LIN {X 0.027,Y -509.372,Z 664.122,A 0.000,B 0.000,C 90.000,E1 237.995} C_DIS
LIN {X 0.006,Y -505.336,Z 664.112,A 0.000,B 0.000,C 90.000,E1 236.215} C_DIS
LIN {X -0.007,Y -502.437,Z 664.106,A 0.000,B 0.000,C 90.000,E1 235.022} C_DIS
LIN {X 0.219,Y -498.643,Z 664.097,A 0.000,B 0.000,C 90.000,E1 233.497} C_DIS
LIN {X -0.007,Y -491.952,Z 664.082,A 0.000,B 0.000,C 90.000,E1 230.803} C_DIS
LIN {X -0.006,Y -487.620,Z 664.072,A 0.000,B 0.000,C 90.000,E1 228.976} C_DIS
LIN {X 0.039,Y -482.507,Z 664.060,A 0.000,B 0.000,C 90.000,E1 226.824} C_DIS
LIN {X 0.020,Y -478.874,Z 664.052,A 0.000,B 0.000,C 90.000,E1 225.283} C_DIS
LIN {X 0.140,Y -473.719,Z 664.040,A 0.000,B 0.000,C 90.000,E1 223.095} C_DIS
LIN {X -0.036,Y -467.402,Z 664.024,A 0.000,B 0.000,C 90.000,E1 220.297} C_DIS
LIN {X 0.130,Y -463.516,Z 664.013,A 0.000,B 0.000,C 90.000,E1 218.382} C_DIS
LIN {X 0.034,Y -459.004,Z 664.001,A 0.000,B 0.000,C 90.000,E1 216.171} C_DIS
LIN {X 0.087,Y -455.266,Z 663.990,A 0.000,B 0.000,C 90.000,E1 214.246} C_DIS
LIN {X 0.106,Y -452.881,Z 663.983,A 0.000,B 0.000,C 90.000,E1 212.959} C_DIS
LIN {X -0.122,Y -449.264,Z 663.972,A 0.000,B 0.000,C 90.000,E1 211.052} C_DIS
LIN {X 0.103,Y -445.713,Z 663.962,A 0.000,B 0.000,C 90.000,E1 209.077} C_DIS
LIN {X -0.017,Y -442.739,Z 663.953,A 0.000,B 0.000,C 90.000,E1 207.462} C_DIS
LIN {X -0.194,Y -439.843,Z 663.943,A 0.000,B 0.000,C 90.000,E1 205.848} C_DIS
LIN {X -0.225,Y -436.925,Z 663.934,A 0.000,B 0.000,C 90.000,E1 204.207} C_DIS
LIN {X -0.094,Y -433.311,Z 663.923,A 0.000,B 0.000,C 90.000,E1 202.206} C_DIS
LIN {X -0.011,Y -429.068,Z 663.910,A 0.000,B 0.000,C 90.000,E1 199.866} C_DIS
LIN {X -0.132,Y -425.619,Z 663.899,A 0.000,B 0.000,C 90.000,E1 197.873} C_DIS
LIN {X -0.234,Y -422.836,Z 663.890,A 0.000,B 0.000,C 90.000,E1 196.205} C_DIS
LIN {X 0.185,Y -419.483,Z 663.879,A 0.000,B 0.000,C 90.000,E1 194.120} C_DIS
LIN {X -0.098,Y -416.086,Z 663.867,A 0.000,B 0.000,C 90.000,E1 192.119} C_DIS
LIN {X -0.141,Y -412.932,Z 663.856,A 0.000,B 0.000,C 90.000,E1 190.074} C_DIS
LIN {X 0.011,Y -409.838,Z 663.844,A 0.000,B 0.000,C 90.000,E1 187.992} C_DIS
LIN {X 0.058,Y -406.301,Z 663.831,A 0.000,B 0.000,C 90.000,E1 185.568} C_DIS
LIN {X -0.081,Y -402.738,Z 663.816,A 0.000,B 0.000,C 90.000,E1 182.808} C_DIS
LIN {X -0.038,Y -399.329,Z 663.798,A 0.000,B 0.000,C 90.000,E1 179.656} C_DIS
LIN {X -0.157,Y -396.563,Z 663.779,A 0.000,B 0.000,C 90.000,E1 176.159} C_DIS
LIN {X 0.204,Y -394.877,Z 663.761,A 0.000,B 0.000,C 90.000,E1 172.932} C_DIS
LIN {X -0.093,Y -394.008,Z 663.747,A 0.000,B 0.000,C 90.000,E1 170.500} C_DIS
LIN {X 0.062,Y -393.548,Z 663.731,A 0.000,B 0.000,C 90.000,E1 167.645} C_DIS
LIN {X 0.067,Y -393.374,Z 663.720,A 0.000,B 0.000,C 90.000,E1 165.519} C_DIS
LIN {X 0.114,Y -393.447,Z 663.706,A 0.000,B 0.000,C 90.000,E1 163.032} C_DIS
LIN {X 0.127,Y -393.772,Z 663.692,A 0.000,B 0.000,C 90.000,E1 160.550} C_DIS
LIN {X -0.021,Y -393.961,Z 663.684,A 0.000,B 0.000,C 90.000,E1 159.156} C_DIS
LIN {X -0.140,Y -394.297,Z 663.672,A 0.000,B 0.000,C 90.000,E1 157.050} C_DIS
LIN {X -0.030,Y -394.820,Z 663.657,A 0.000,B 0.000,C 90.000,E1 154.204} C_DIS
LIN {X 0.159,Y -395.196,Z 663.647,A 0.000,B 0.000,C 90.000,E1 152.410} C_DIS
LIN {X -0.136,Y -395.685,Z 663.635,A 0.000,B 0.000,C 90.000,E1 150.333} C_DIS
LIN {X -0.161,Y -396.344,Z 663.621,A 0.000,B 0.000,C 90.000,E1 147.867} C_DIS
LIN {X -0.079,Y -397.264,Z 663.608,A 0.000,B 0.000,C 90.000,E1 145.388} C_DIS
LIN {X 0.066,Y -398.259,Z 663.596,A 0.000,B 0.000,C 90.000,E1 143.256} C_DIS
LIN {X -0.084,Y -399.368,Z 663.584,A 0.000,B 0.000,C 90.000,E1 141.170} C_DIS
LIN {X 0.099,Y -400.918,Z 663.571,A 0.000,B 0.000,C 90.000,E1 138.690} C_DIS
LIN {X -0.036,Y -401.754,Z 663.563,A 0.000,B 0.000,C 90.000,E1 137.310} C_DIS
LIN {X 0.162,Y -403.361,Z 663.549,A 0.000,B 0.000,C 90.000,E1 134.838} C_DIS
LIN {X -0.124,Y -404.797,Z 663.540,A 0.000,B 0.000,C 90.000,E1 133.137} C_DIS
LIN {X -0.166,Y -405.700,Z 663.536,A 0.000,B 0.000,C 90.000,E1 132.447} C_DIS
LIN {X -0.200,Y -406.988,Z 663.532,A 0.000,B 0.000,C 90.000,E1 131.757} C_DIS
LIN {X -0.183,Y -409.105,Z 663.529,A 0.000,B 0.000,C 90.000,E1 131.148} C_DIS
LIN {X -0.042,Y -411.236,Z 663.527,A 0.000,B 0.000,C 90.000,E1 130.782} C_DIS
LIN {X -0.120,Y -412.190,Z 663.526,A 0.000,B 0.000,C 90.000,E1 130.620} C_DIS
LIN {X -0.196,Y -413.918,Z 663.525,A 0.000,B 0.000,C 90.000,E1 130.458} C_DIS
LIN {X 0.055,Y -417.079,Z 663.523,A 0.000,B 0.000,C 90.000,E1 130.092} C_DIS
LIN {X -0.146,Y -423.546,Z 663.520,A 0.000,B 0.000,C 90.000,E1 129.564} C_DIS
LIN {X 0.122,Y -449.130,Z 663.509,A 0.000,B 0.000,C 90.000,E1 127.604} C_DIS
LIN {X 0.249,Y -459.985,Z 663.505,A 0.000,B 0.000,C 90.000,E1 126.790} C_DIS
LIN {X 0.184,Y -467.766,Z 663.501,A 0.000,B 0.000,C 90.000,E1 126.217} C_DIS
LIN {X 0.030,Y -473.899,Z 663.499,A 0.000,B 0.000,C 90.000,E1 125.758} C_DIS
LIN {X 0.100,Y -481.253,Z 663.495,A 0.000,B 0.000,C 90.000,E1 125.152} C_DIS
LIN {X -0.243,Y -485.709,Z 663.493,A 0.000,B 0.000,C 90.000,E1 124.818} C_DIS
LIN {X 0.011,Y -491.516,Z 663.490,A 0.000,B 0.000,C 90.000,E1 124.278} C_DIS
LIN {X 0.140,Y -500.006,Z 663.486,A 0.000,B 0.000,C 90.000,E1 123.499} C_DIS
LIN {X -0.253,Y -509.537,Z 663.481,A 0.000,B 0.000,C 90.000,E1 122.625} C_DIS
LIN {X -0.014,Y -515.907,Z 663.478,A 0.000,B 0.000,C 90.000,E1 121.957} C_DIS
LIN {X 0.036,Y -523.749,Z 663.473,A 0.000,B 0.000,C 90.000,E1 121.131} C_DIS
LIN {X -0.228,Y -528.777,Z 663.470,A 0.000,B 0.000,C 90.000,E1 120.590} C_DIS
LIN {X -0.159,Y -533.124,Z 663.467,A 0.000,B 0.000,C 90.000,E1 120.050} C_DIS
LIN {X -0.017,Y -537.366,Z 663.464,A 0.000,B 0.000,C 90.000,E1 119.461} C_DIS
LIN {X 0.025,Y -542.151,Z 663.460,A 0.000,B 0.000,C 90.000,E1 118.743} C_DIS
LIN {X 0.114,Y -546.377,Z 663.456,A 0.000,B 0.000,C 90.000,E1 118.025} C_DIS
LIN {X 0.105,Y -549.500,Z 663.453,A 0.000,B 0.000,C 90.000,E1 117.462} C_DIS
LIN {X 0.147,Y -553.631,Z 663.448,A 0.000,B 0.000,C 90.000,E1 116.616} C_DIS
LIN {X 0.091,Y -556.868,Z 663.444,A 0.000,B 0.000,C 90.000,E1 115.924} C_DIS
LIN {X 0.197,Y -560.328,Z 663.440,A 0.000,B 0.000,C 90.000,E1 115.079} C_DIS
LIN {X -0.103,Y -564.545,Z 663.433,A 0.000,B 0.000,C 90.000,E1 114.003} C_DIS
LIN {X -0.054,Y -568.273,Z 663.427,A 0.000,B 0.000,C 90.000,E1 112.898} C_DIS
LIN {X -0.078,Y -570.823,Z 663.423,A 0.000,B 0.000,C 90.000,E1 112.078} C_DIS
LIN {X -0.116,Y -572.382,Z 663.420,A 0.000,B 0.000,C 90.000,E1 111.535} C_DIS
LIN {X 0.054,Y -575.058,Z 663.414,A 0.000,B 0.000,C 90.000,E1 110.429} C_DIS
LIN {X 0.258,Y -577.513,Z 663.408,A 0.000,B 0.000,C 90.000,E1 109.322} C_DIS
LIN {X 0.302,Y -579.804,Z 663.402,A 0.000,B 0.000,C 90.000,E1 108.236} C_DIS
LIN {X -0.080,Y -583.716,Z 663.391,A 0.000,B 0.000,C 90.000,E1 106.386} C_DIS
LIN {X 0.281,Y -586.439,Z 663.384,A 0.000,B 0.000,C 90.000,E1 105.009} C_DIS
LIN {X -0.041,Y -589.129,Z 663.376,A 0.000,B 0.000,C 90.000,E1 103.703} C_DIS
LIN {X -0.151,Y -591.244,Z 663.370,A 0.000,B 0.000,C 90.000,E1 102.647} C_DIS
LIN {X 0.183,Y -595.368,Z 663.358,A 0.000,B 0.000,C 90.000,E1 100.489} C_DIS
LIN {X 0.046,Y -598.366,Z 663.350,A 0.000,B 0.000,C 90.000,E1 98.916} C_DIS
LIN {X -0.053,Y -600.257,Z 663.344,A 0.000,B 0.000,C 90.000,E1 97.871} C_DIS
LIN {X 0.022,Y -602.401,Z 663.336,A 0.000,B 0.000,C 90.000,E1 96.549} C_DIS
LIN {X 0.262,Y -603.616,Z 663.332,A 0.000,B 0.000,C 90.000,E1 95.739} C_DIS
LIN {X -0.197,Y -605.551,Z 663.325,A 0.000,B 0.000,C 90.000,E1 94.473} C_DIS
LIN {X -0.062,Y -607.203,Z 663.318,A 0.000,B 0.000,C 90.000,E1 93.154} C_DIS
LIN {X 0.108,Y -608.659,Z 663.310,A 0.000,B 0.000,C 90.000,E1 91.835} C_DIS
LIN {X 0.296,Y -609.771,Z 663.303,A 0.000,B 0.000,C 90.000,E1 90.516} C_DIS
LIN {X 0.205,Y -610.431,Z 663.297,A 0.000,B 0.000,C 90.000,E1 89.484} C_DIS
LIN {X 0.118,Y -610.892,Z 663.292,A 0.000,B 0.000,C 90.000,E1 88.453} C_DIS
LIN {X 0.054,Y -611.171,Z 663.286,A 0.000,B 0.000,C 90.000,E1 87.421} C_DIS
LIN {X -0.001,Y -611.342,Z 663.280,A 0.000,B 0.000,C 90.000,E1 86.388} C_DIS
LIN {X -0.058,Y -611.310,Z 663.274,A 0.000,B 0.000,C 90.000,E1 85.355} C_DIS
LIN {X 0.205,Y -610.994,Z 663.267,A 0.000,B 0.000,C 90.000,E1 84.033} C_DIS
LIN {X 0.191,Y -610.576,Z 663.261,A 0.000,B 0.000,C 90.000,E1 82.996} C_DIS
LIN {X 0.253,Y -610.067,Z 663.255,A 0.000,B 0.000,C 90.000,E1 81.951} C_DIS
LIN {X 0.219,Y -609.190,Z 663.250,A 0.000,B 0.000,C 90.000,E1 80.914} C_DIS
LIN {X 0.031,Y -608.443,Z 663.245,A 0.000,B 0.000,C 90.000,E1 80.151} C_DIS
LIN {X -0.193,Y -606.957,Z 663.238,A 0.000,B 0.000,C 90.000,E1 78.870} C_DIS
LIN {X 0.271,Y -605.274,Z 663.231,A 0.000,B 0.000,C 90.000,E1 77.521} C_DIS
LIN {X -0.204,Y -603.788,Z 663.225,A 0.000,B 0.000,C 90.000,E1 76.520} C_DIS
LIN {X 0.193,Y -601.761,Z 663.218,A 0.000,B 0.000,C 90.000,E1 75.172} C_DIS
LIN {X 0.099,Y -600.497,Z 663.213,A 0.000,B 0.000,C 90.000,E1 74.393} C_DIS
LIN {X 0.288,Y -598.679,Z 663.208,A 0.000,B 0.000,C 90.000,E1 73.323} C_DIS
LIN {X -0.127,Y -596.729,Z 663.202,A 0.000,B 0.000,C 90.000,E1 72.308} C_DIS
LIN {X 0.179,Y -594.711,Z 663.196,A 0.000,B 0.000,C 90.000,E1 71.221} C_DIS
LIN {X -0.216,Y -591.898,Z 663.188,A 0.000,B 0.000,C 90.000,E1 69.934} C_DIS
LIN {X 0.015,Y -589.281,Z 663.183,A 0.000,B 0.000,C 90.000,E1 68.847} C_DIS
LIN {X -0.011,Y -587.181,Z 663.178,A 0.000,B 0.000,C 90.000,E1 68.050} C_DIS
LIN {X 0.165,Y -584.852,Z 663.174,A 0.000,B 0.000,C 90.000,E1 67.230} C_DIS
LIN {X -0.042,Y -581.402,Z 663.168,A 0.000,B 0.000,C 90.000,E1 66.177} C_DIS
LIN {X 0.079,Y -578.533,Z 663.163,A 0.000,B 0.000,C 90.000,E1 65.357} C_DIS
LIN {X 0.169,Y -575.542,Z 663.159,A 0.000,B 0.000,C 90.000,E1 64.537} C_DIS
LIN {X 0.064,Y -571.154,Z 663.153,A 0.000,B 0.000,C 90.000,E1 63.461} C_DIS
LIN {X -0.008,Y -568.900,Z 663.150,A 0.000,B 0.000,C 90.000,E1 62.922} C_DIS
LIN {X -0.025,Y -565.254,Z 663.145,A 0.000,B 0.000,C 90.000,E1 62.103} C_DIS
LIN {X 0.268,Y -561.861,Z 663.141,A 0.000,B 0.000,C 90.000,E1 61.385} C_DIS
LIN {X 0.223,Y -558.151,Z 663.138,A 0.000,B 0.000,C 90.000,E1 60.717} C_DIS
LIN {X -0.031,Y -553.887,Z 663.134,A 0.000,B 0.000,C 90.000,E1 60.049} C_DIS
LIN {X -0.007,Y -550.136,Z 663.131,A 0.000,B 0.000,C 90.000,E1 59.488} C_DIS
LIN {X -0.207,Y -546.031,Z 663.127,A 0.000,B 0.000,C 90.000,E1 58.948} C_DIS
LIN {X -0.029,Y -540.656,Z 663.124,A 0.000,B 0.000,C 90.000,E1 58.280} C_DIS
LIN {X -0.246,Y -535.968,Z 663.121,A 0.000,B 0.000,C 90.000,E1 57.788} C_DIS
LIN {X 0.095,Y -530.631,Z 663.118,A 0.000,B 0.000,C 90.000,E1 57.248} C_DIS
LIN {X 0.012,Y -524.965,Z 663.116,A 0.000,B 0.000,C 90.000,E1 56.786} C_DIS
LIN {X 0.049,Y -520.270,Z 663.114,A 0.000,B 0.000,C 90.000,E1 56.421} C_DIS
LIN {X 0.038,Y -515.339,Z 663.112,A 0.000,B 0.000,C 90.000,E1 56.087} C_DIS
LIN {X 0.084,Y -508.668,Z 663.109,A 0.000,B 0.000,C 90.000,E1 55.674} C_DIS
LIN {X 0.283,Y -500.535,Z 663.107,A 0.000,B 0.000,C 90.000,E1 55.182} C_DIS
LIN {X 0.242,Y -482.123,Z 663.101,A 0.000,B 0.000,C 90.000,E1 54.196} C_DIS
LIN {X 0.109,Y -463.687,Z 663.096,A 0.000,B 0.000,C 90.000,E1 53.210} C_DIS
LIN {X 0.025,Y -433.343,Z 663.086,A 0.000,B 0.000,C 90.000,E1 51.457} C_DIS
LIN {X 0.006,Y -432.617,Z 663.086,A 0.000,B 0.000,C 90.000,E1 51.412} C_DIS
LIN {X -0.018,Y -432.584,Z 663.086,A 0.000,B 0.000,C 90.000,E1 51.412} C_DIS
LIN {X 0.025,Y -431.721,Z 663.083,A 0.000,B 0.000,C 90.000,E1 50.928} C_DIS
LIN {X -0.067,Y -430.119,Z 663.079,A 0.000,B 0.000,C 90.000,E1 50.275} C_DIS
LIN {X 0.066,Y -420.564,Z 663.055,A 0.000,B 0.000,C 90.000,E1 45.891} C_DIS
LIN {X -0.047,Y -418.253,Z 663.048,A 0.000,B 0.000,C 90.000,E1 44.636} C_DIS
LIN {X -0.178,Y -418.393,Z 663.036,A 0.000,B 0.000,C 90.000,E1 42.528} C_DIS
LIN {X 0.234,Y -418.755,Z 663.023,A 0.000,B 0.000,C 90.000,E1 40.092} C_DIS
LIN {X -0.071,Y -419.790,Z 663.006,A 0.000,B 0.000,C 90.000,E1 37.076} C_DIS
LIN {X 0.009,Y -421.040,Z 662.993,A 0.000,B 0.000,C 90.000,E1 34.692} C_DIS
LIN {X -0.116,Y -422.242,Z 662.980,A 0.000,B 0.000,C 90.000,E1 32.339} C_DIS
LIN {X -0.203,Y -422.780,Z 662.974,A 0.000,B 0.000,C 90.000,E1 31.337} C_DIS
LIN {X 0.013,Y -423.850,Z 662.963,A 0.000,B 0.000,C 90.000,E1 29.283} C_DIS
LIN {X 0.046,Y -425.021,Z 662.952,A 0.000,B 0.000,C 90.000,E1 27.257} C_DIS
LIN {X 0.028,Y -427.312,Z 662.933,A 0.000,B 0.000,C 90.000,E1 23.898} C_DIS
LIN {X 0.167,Y -429.397,Z 662.920,A 0.000,B 0.000,C 90.000,E1 21.535} C_DIS
LIN {X -0.196,Y -430.627,Z 662.912,A 0.000,B 0.000,C 90.000,E1 20.248} C_DIS
LIN {X 0.082,Y -431.830,Z 662.903,A 0.000,B 0.000,C 90.000,E1 18.544} C_DIS
LIN {X 0.159,Y -433.396,Z 662.890,A 0.000,B 0.000,C 90.000,E1 16.205} C_DIS
LIN {X 0.154,Y -435.232,Z 662.877,A 0.000,B 0.000,C 90.000,E1 13.883} C_DIS
LIN {X -0.244,Y -437.067,Z 662.866,A 0.000,B 0.000,C 90.000,E1 11.951} C_DIS
LIN {X 0.124,Y -439.711,Z 662.852,A 0.000,B 0.000,C 90.000,E1 9.265} C_DIS
LIN {X -0.067,Y -442.666,Z 662.837,A 0.000,B 0.000,C 90.000,E1 6.663} C_DIS
LIN {X -0.073,Y -445.063,Z 662.826,A 0.000,B 0.000,C 90.000,E1 4.702} C_DIS
LIN {X 0.043,Y -448.179,Z 662.813,A 0.000,B 0.000,C 90.000,E1 2.407} C_DIS
LIN {X 0.220,Y -453.617,Z 662.794,A 0.000,B 0.000,C 90.000,E1 358.797} C_DIS
LIN {X 0.200,Y -456.324,Z 662.785,A 0.000,B 0.000,C 90.000,E1 357.192} C_DIS
LIN {X 0.213,Y -460.314,Z 662.772,A 0.000,B 0.000,C 90.000,E1 354.951} C_DIS
LIN {X 0.129,Y -463.792,Z 662.762,A 0.000,B 0.000,C 90.000,E1 353.053} C_DIS
LIN {X 0.236,Y -467.256,Z 662.751,A 0.000,B 0.000,C 90.000,E1 351.141} C_DIS
LIN {X 0.141,Y -470.056,Z 662.742,A 0.000,B 0.000,C 90.000,E1 349.577} C_DIS
LIN {X -0.019,Y -472.273,Z 662.735,A 0.000,B 0.000,C 90.000,E1 348.342} C_DIS
LIN {X 0.000,Y -475.632,Z 662.725,A 0.000,B 0.000,C 90.000,E1 346.464} C_DIS
LIN {X -0.228,Y -478.519,Z 662.716,A 0.000,B 0.000,C 90.000,E1 344.936} C_DIS
LIN {X 0.156,Y -482.061,Z 662.706,A 0.000,B 0.000,C 90.000,E1 343.032} C_DIS
LIN {X -0.150,Y -486.282,Z 662.694,A 0.000,B 0.000,C 90.000,E1 340.913} C_DIS
LIN {X -0.202,Y -489.942,Z 662.684,A 0.000,B 0.000,C 90.000,E1 339.082} C_DIS
LIN {X -0.073,Y -492.394,Z 662.677,A 0.000,B 0.000,C 90.000,E1 337.847} C_DIS
LIN {X 0.137,Y -495.253,Z 662.669,A 0.000,B 0.000,C 90.000,E1 336.305} C_DIS
LIN {X 0.034,Y -496.856,Z 662.663,A 0.000,B 0.000,C 90.000,E1 335.409} C_DIS
LIN {X -0.038,Y -500.553,Z 662.652,A 0.000,B 0.000,C 90.000,E1 333.307} C_DIS
LIN {X 0.289,Y -503.556,Z 662.643,A 0.000,B 0.000,C 90.000,E1 331.769} C_DIS
LIN {X 0.214,Y -505.139,Z 662.640,A 0.000,B 0.000,C 90.000,E1 331.179} C_DIS
LIN {X -0.164,Y -506.086,Z 662.638,A 0.000,B 0.000,C 90.000,E1 330.923} C_DIS
LIN {X -0.035,Y -507.866,Z 662.636,A 0.000,B 0.000,C 90.000,E1 330.461} C_DIS
LIN {X 0.288,Y -509.367,Z 662.634,A 0.000,B 0.000,C 90.000,E1 330.127} C_DIS
LIN {X 0.087,Y -511.675,Z 662.632,A 0.000,B 0.000,C 90.000,E1 329.822} C_DIS
LIN {X -0.121,Y -515.763,Z 662.630,A 0.000,B 0.000,C 90.000,E1 329.410} C_DIS
LIN {X 0.038,Y -517.228,Z 662.629,A 0.000,B 0.000,C 90.000,E1 329.253} C_DIS
LIN {X -0.049,Y -528.261,Z 662.625,A 0.000,B 0.000,C 90.000,E1 328.408} C_DIS
LIN {X -0.019,Y -535.587,Z 662.622,A 0.000,B 0.000,C 90.000,E1 327.867} C_DIS
LIN {X -0.005,Y -542.881,Z 662.618,A 0.000,B 0.000,C 90.000,E1 327.296} C_DIS
LIN {X -0.047,Y -549.996,Z 662.615,A 0.000,B 0.000,C 90.000,E1 326.707} C_DIS
LIN {X 0.101,Y -557.016,Z 662.612,A 0.000,B 0.000,C 90.000,E1 326.087} C_DIS
LIN {X 0.044,Y -563.819,Z 662.608,A 0.000,B 0.000,C 90.000,E1 325.468} C_DIS
LIN {X -0.216,Y -574.514,Z 662.603,A 0.000,B 0.000,C 90.000,E1 324.482} C_DIS
LIN {X -0.068,Y -583.656,Z 662.598,A 0.000,B 0.000,C 90.000,E1 323.577} C_DIS
LIN {X 0.117,Y -588.789,Z 662.595,A 0.000,B 0.000,C 90.000,E1 323.050} C_DIS
LIN {X -0.028,Y -598.878,Z 662.589,A 0.000,B 0.000,C 90.000,E1 322.029} C_DIS
LIN {X -0.187,Y -603.647,Z 662.586,A 0.000,B 0.000,C 90.000,E1 321.537} C_DIS
LIN {X -0.202,Y -609.452,Z 662.583,A 0.000,B 0.000,C 90.000,E1 320.884} C_DIS
LIN {X 0.221,Y -614.894,Z 662.579,A 0.000,B 0.000,C 90.000,E1 320.194} C_DIS
LIN {X 0.303,Y -619.990,Z 662.575,A 0.000,B 0.000,C 90.000,E1 319.542} C_DIS
LIN {X 0.319,Y -625.551,Z 662.571,A 0.000,B 0.000,C 90.000,E1 318.771} C_DIS
LIN {X -0.028,Y -630.814,Z 662.567,A 0.000,B 0.000,C 90.000,E1 318.038} C_DIS
LIN {X 0.022,Y -636.642,Z 662.562,A 0.000,B 0.000,C 90.000,E1 317.148} C_DIS
LIN {X -0.374,Y -643.605,Z 662.556,A 0.000,B 0.000,C 90.000,E1 316.053} C_DIS
LIN {X 0.266,Y -649.520,Z 662.550,A 0.000,B 0.000,C 90.000,E1 315.000} C_DIS
LIN {X 0.068,Y -655.214,Z 662.545,A 0.000,B 0.000,C 90.000,E1 314.028} C_DIS
LIN {X -0.091,Y -661.642,Z 662.538,A 0.000,B 0.000,C 90.000,E1 312.813} C_DIS
LIN {X 0.357,Y -667.076,Z 662.532,A 0.000,B 0.000,C 90.000,E1 311.676} C_DIS
LIN {X -0.095,Y -671.643,Z 662.526,A 0.000,B 0.000,C 90.000,E1 310.744} C_DIS
LIN {X 0.016,Y -675.774,Z 662.521,A 0.000,B 0.000,C 90.000,E1 309.769} C_DIS
LIN {X 0.157,Y -678.572,Z 662.517,A 0.000,B 0.000,C 90.000,E1 309.036} C_DIS
LIN {X -0.068,Y -681.895,Z 662.512,A 0.000,B 0.000,C 90.000,E1 308.096} C_DIS
LIN {X 0.136,Y -684.187,Z 662.508,A 0.000,B 0.000,C 90.000,E1 307.363} C_DIS
LIN {X -0.020,Y -687.018,Z 662.502,A 0.000,B 0.000,C 90.000,E1 306.423} C_DIS
LIN {X 0.013,Y -689.561,Z 662.497,A 0.000,B 0.000,C 90.000,E1 305.471} C_DIS
LIN {X -0.082,Y -691.916,Z 662.492,A 0.000,B 0.000,C 90.000,E1 304.532} C_DIS
LIN {X 0.027,Y -694.069,Z 662.487,A 0.000,B 0.000,C 90.000,E1 303.579} C_DIS
LIN {X 0.170,Y -696.000,Z 662.481,A 0.000,B 0.000,C 90.000,E1 302.625} C_DIS
LIN {X 0.338,Y -697.768,Z 662.476,A 0.000,B 0.000,C 90.000,E1 301.671} C_DIS
LIN {X -0.178,Y -699.731,Z 662.470,A 0.000,B 0.000,C 90.000,E1 300.541} C_DIS
LIN {X 0.362,Y -700.743,Z 662.466,A 0.000,B 0.000,C 90.000,E1 299.795} C_DIS
LIN {X -0.122,Y -702.115,Z 662.459,A 0.000,B 0.000,C 90.000,E1 298.665} C_DIS
LIN {X 0.038,Y -703.130,Z 662.454,A 0.000,B 0.000,C 90.000,E1 297.719} C_DIS
LIN {X -0.114,Y -704.276,Z 662.448,A 0.000,B 0.000,C 90.000,E1 296.565} C_DIS
LIN {X -0.171,Y -704.660,Z 662.445,A 0.000,B 0.000,C 90.000,E1 296.104} C_DIS
LIN {X 0.404,Y -704.890,Z 662.442,A 0.000,B 0.000,C 90.000,E1 295.591} C_DIS
LIN {X 0.041,Y -704.354,Z 662.440,A 0.000,B 0.000,C 90.000,E1 295.155} C_DIS
LIN {X 0.327,Y -703.975,Z 662.439,A 0.000,B 0.000,C 90.000,E1 294.899} C_DIS
LIN {X -0.178,Y -702.250,Z 662.437,A 0.000,B 0.000,C 90.000,E1 294.591} C_DIS
LIN {X 0.240,Y -700.099,Z 662.435,A 0.000,B 0.000,C 90.000,E1 294.207} C_DIS
LIN {X 0.376,Y -698.957,Z 662.434,A 0.000,B 0.000,C 90.000,E1 294.079} C_DIS
LIN {X -0.030,Y -695.643,Z 662.433,A 0.000,B 0.000,C 90.000,E1 293.898} C_DIS
LIN {X 0.171,Y -692.436,Z 662.432,A 0.000,B 0.000,C 90.000,E1 293.695} C_DIS
LIN {X -0.285,Y -690.675,Z 662.431,A 0.000,B 0.000,C 90.000,E1 293.643} C_DIS
LIN {X 0.287,Y -688.082,Z 662.431,A 0.000,B 0.000,C 90.000,E1 293.515} C_DIS
LIN {X -0.024,Y -680.661,Z 662.430,A 0.000,B 0.000,C 90.000,E1 293.387} C_DIS
LIN {X 0.053,Y -670.907,Z 662.429,A 0.000,B 0.000,C 90.000,E1 293.259} C_DIS
LIN {X -0.245,Y -663.165,Z 662.429,A 0.000,B 0.000,C 90.000,E1 293.206} C_DIS
LIN {X -0.108,Y -649.981,Z 662.428,A 0.000,B 0.000,C 90.000,E1 293.003} C_DIS
LIN {X -0.121,Y -640.326,Z 662.427,A 0.000,B 0.000,C 90.000,E1 292.823} C_DIS
LIN {X 0.020,Y -629.959,Z 662.426,A 0.000,B 0.000,C 90.000,E1 292.589} C_DIS
LIN {X 0.081,Y -613.500,Z 662.423,A 0.000,B 0.000,C 90.000,E1 292.153} C_DIS
LIN {X 0.017,Y -579.129,Z 662.417,A 0.000,B 0.000,C 90.000,E1 291.099} C_DIS
LIN {X -0.131,Y -563.252,Z 662.415,A 0.000,B 0.000,C 90.000,E1 290.663} C_DIS
LIN {X -0.179,Y -559.151,Z 662.414,A 0.000,B 0.000,C 90.000,E1 290.482} C_DIS
LIN {X 0.083,Y -556.206,Z 662.413,A 0.000,B 0.000,C 90.000,E1 290.301} C_DIS
LIN {X 0.041,Y -556.157,Z 662.413,A 0.000,B 0.000,C 90.000,E1 290.301} C_DIS
LIN {X 0.108,Y -555.403,Z 662.412,A 0.000,B 0.000,C 90.000,E1 290.174} C_DIS
LIN {X 0.034,Y -554.964,Z 662.411,A 0.000,B 0.000,C 90.000,E1 289.885} C_DIS
LIN {X 0.085,Y -554.601,Z 662.407,A 0.000,B 0.000,C 90.000,E1 289.322} C_DIS
LIN {X -0.195,Y -554.511,Z 662.401,A 0.000,B 0.000,C 90.000,E1 288.236} C_DIS
LIN {X -0.093,Y -554.079,Z 662.392,A 0.000,B 0.000,C 90.000,E1 286.551} C_DIS
LIN {X 0.108,Y -553.584,Z 662.384,A 0.000,B 0.000,C 90.000,E1 285.134} C_DIS
LIN {X 0.192,Y -553.105,Z 662.378,A 0.000,B 0.000,C 90.000,E1 284.008} C_DIS
LIN {X 0.082,Y -552.036,Z 662.367,A 0.000,B 0.000,C 90.000,E1 282.063} C_DIS
LIN {X -0.283,Y -551.106,Z 662.356,A 0.000,B 0.000,C 90.000,E1 280.141} C_DIS
LIN {X -0.127,Y -550.431,Z 662.345,A 0.000,B 0.000,C 90.000,E1 278.163} C_DIS
LIN {X -0.147,Y -549.997,Z 662.334,A 0.000,B 0.000,C 90.000,E1 276.201} C_DIS
LIN {X -0.143,Y -549.689,Z 662.322,A 0.000,B 0.000,C 90.000,E1 273.955} C_DIS
LIN {X 0.086,Y -549.475,Z 662.316,A 0.000,B 0.000,C 90.000,E1 272.808} C_DIS
LIN {X -0.236,Y -549.182,Z 662.309,A 0.000,B 0.000,C 90.000,E1 271.718} C_DIS
LIN {X 0.022,Y -548.566,Z 662.302,A 0.000,B 0.000,C 90.000,E1 270.286} C_DIS
LIN {X 0.224,Y -548.035,Z 662.295,A 0.000,B 0.000,C 90.000,E1 269.141} C_DIS
LIN {X -0.071,Y -547.233,Z 662.288,A 0.000,B 0.000,C 90.000,E1 267.764} C_DIS
LIN {X 0.204,Y -546.287,Z 662.278,A 0.000,B 0.000,C 90.000,E1 266.045} C_DIS
LIN {X -0.093,Y -545.187,Z 662.270,A 0.000,B 0.000,C 90.000,E1 264.666} C_DIS
LIN {X 0.110,Y -544.261,Z 662.264,A 0.000,B 0.000,C 90.000,E1 263.514} C_DIS
LIN {X -0.167,Y -542.784,Z 662.256,A 0.000,B 0.000,C 90.000,E1 262.129} C_DIS
LIN {X 0.067,Y -541.603,Z 662.250,A 0.000,B 0.000,C 90.000,E1 260.971} C_DIS
LIN {X 0.108,Y -539.197,Z 662.236,A 0.000,B 0.000,C 90.000,E1 258.409} C_DIS
LIN {X 0.168,Y -537.484,Z 662.225,A 0.000,B 0.000,C 90.000,E1 256.408} C_DIS
LIN {X 0.019,Y -536.557,Z 662.218,A 0.000,B 0.000,C 90.000,E1 255.283} C_DIS
LIN {X -0.143,Y -535.539,Z 662.212,A 0.000,B 0.000,C 90.000,E1 254.157} C_DIS
LIN {X 0.065,Y -533.824,Z 662.202,A 0.000,B 0.000,C 90.000,E1 252.417} C_DIS
LIN {X -0.274,Y -532.128,Z 662.193,A 0.000,B 0.000,C 90.000,E1 250.732} C_DIS
LIN {X -0.179,Y -530.804,Z 662.186,A 0.000,B 0.000,C 90.000,E1 249.571} C_DIS
LIN {X -0.228,Y -528.367,Z 662.177,A 0.000,B 0.000,C 90.000,E1 247.847} C_DIS
LIN {X -0.171,Y -527.108,Z 662.172,A 0.000,B 0.000,C 90.000,E1 246.975} C_DIS
LIN {X -0.128,Y -525.770,Z 662.167,A 0.000,B 0.000,C 90.000,E1 246.102} C_DIS
LIN {X -0.255,Y -523.193,Z 662.159,A 0.000,B 0.000,C 90.000,E1 244.665} C_DIS
LIN {X -0.038,Y -521.614,Z 662.154,A 0.000,B 0.000,C 90.000,E1 243.768} C_DIS
LIN {X -0.165,Y -519.271,Z 662.148,A 0.000,B 0.000,C 90.000,E1 242.615} C_DIS
LIN {X 0.035,Y -516.270,Z 662.140,A 0.000,B 0.000,C 90.000,E1 241.129} C_DIS
LIN {X -0.023,Y -513.089,Z 662.132,A 0.000,B 0.000,C 90.000,E1 239.665} C_DIS
LIN {X 0.199,Y -509.109,Z 662.122,A 0.000,B 0.000,C 90.000,E1 237.867} C_DIS
LIN {X -0.148,Y -505.754,Z 662.113,A 0.000,B 0.000,C 90.000,E1 236.421} C_DIS
LIN {X 0.259,Y -502.855,Z 662.107,A 0.000,B 0.000,C 90.000,E1 235.182} C_DIS
LIN {X 0.085,Y -499.051,Z 662.098,A 0.000,B 0.000,C 90.000,E1 233.703} C_DIS
LIN {X -0.122,Y -492.319,Z 662.083,A 0.000,B 0.000,C 90.000,E1 231.009} C_DIS
LIN {X 0.096,Y -487.285,Z 662.072,A 0.000,B 0.000,C 90.000,E1 228.852} C_DIS
LIN {X -0.016,Y -482.911,Z 662.061,A 0.000,B 0.000,C 90.000,E1 227.025} C_DIS
LIN {X -0.041,Y -479.281,Z 662.053,A 0.000,B 0.000,C 90.000,E1 225.486} C_DIS
LIN {X 0.082,Y -474.104,Z 662.041,A 0.000,B 0.000,C 90.000,E1 223.299} C_DIS
LIN {X 0.265,Y -467.745,Z 662.025,A 0.000,B 0.000,C 90.000,E1 220.458} C_DIS
LIN {X 0.077,Y -463.862,Z 662.014,A 0.000,B 0.000,C 90.000,E1 218.588} C_DIS
LIN {X 0.128,Y -460.565,Z 662.006,A 0.000,B 0.000,C 90.000,E1 216.996} C_DIS
LIN {X -0.049,Y -456.797,Z 661.995,A 0.000,B 0.000,C 90.000,E1 215.105} C_DIS
LIN {X -0.029,Y -453.805,Z 661.986,A 0.000,B 0.000,C 90.000,E1 213.499} C_DIS
LIN {X 0.149,Y -450.177,Z 661.975,A 0.000,B 0.000,C 90.000,E1 211.544} C_DIS
LIN {X 0.086,Y -446.019,Z 661.963,A 0.000,B 0.000,C 90.000,E1 209.283} C_DIS
LIN {X 0.028,Y -442.476,Z 661.952,A 0.000,B 0.000,C 90.000,E1 207.334} C_DIS
LIN {X 0.272,Y -439.001,Z 661.941,A 0.000,B 0.000,C 90.000,E1 205.335} C_DIS
LIN {X 0.043,Y -436.006,Z 661.932,A 0.000,B 0.000,C 90.000,E1 203.718} C_DIS
LIN {X -0.069,Y -433.020,Z 661.923,A 0.000,B 0.000,C 90.000,E1 202.078} C_DIS
LIN {X 0.046,Y -429.409,Z 661.912,A 0.000,B 0.000,C 90.000,E1 200.066} C_DIS
LIN {X 0.077,Y -425.929,Z 661.900,A 0.000,B 0.000,C 90.000,E1 198.055} C_DIS
LIN {X -0.020,Y -423.145,Z 661.891,A 0.000,B 0.000,C 90.000,E1 196.386} C_DIS
LIN {X 0.002,Y -419.821,Z 661.880,A 0.000,B 0.000,C 90.000,E1 194.356} C_DIS
LIN {X 0.136,Y -416.432,Z 661.868,A 0.000,B 0.000,C 90.000,E1 192.299} C_DIS
LIN {X 0.105,Y -413.275,Z 661.857,A 0.000,B 0.000,C 90.000,E1 190.254} C_DIS
LIN {X -0.109,Y -410.711,Z 661.848,A 0.000,B 0.000,C 90.000,E1 188.568} C_DIS
LIN {X -0.031,Y -408.133,Z 661.838,A 0.000,B 0.000,C 90.000,E1 186.834} C_DIS
LIN {X -0.116,Y -403.888,Z 661.821,A 0.000,B 0.000,C 90.000,E1 183.726} C_DIS
LIN {X 0.064,Y -401.028,Z 661.807,A 0.000,B 0.000,C 90.000,E1 181.260} C_DIS
LIN {X -0.058,Y -397.510,Z 661.786,A 0.000,B 0.000,C 90.000,E1 177.421} C_DIS
LIN {X -0.095,Y -395.732,Z 661.770,A 0.000,B 0.000,C 90.000,E1 174.609} C_DIS
LIN {X -0.078,Y -394.530,Z 661.754,A 0.000,B 0.000,C 90.000,E1 171.781} C_DIS
LIN {X 0.012,Y -393.733,Z 661.735,A 0.000,B 0.000,C 90.000,E1 168.229} C_DIS
LIN {X -0.070,Y -393.533,Z 661.723,A 0.000,B 0.000,C 90.000,E1 166.117} C_DIS
LIN {X 0.091,Y -393.577,Z 661.709,A 0.000,B 0.000,C 90.000,E1 163.614} C_DIS
LIN {X -0.003,Y -393.849,Z 661.695,A 0.000,B 0.000,C 90.000,E1 161.148} C_DIS
LIN {X -0.086,Y -394.143,Z 661.685,A 0.000,B 0.000,C 90.000,E1 159.390} C_DIS
LIN {X -0.142,Y -394.550,Z 661.672,A 0.000,B 0.000,C 90.000,E1 156.922} C_DIS
LIN {X -0.020,Y -395.099,Z 661.656,A 0.000,B 0.000,C 90.000,E1 154.076} C_DIS
LIN {X 0.173,Y -395.484,Z 661.646,A 0.000,B 0.000,C 90.000,E1 152.281} C_DIS
LIN {X -0.117,Y -395.979,Z 661.634,A 0.000,B 0.000,C 90.000,E1 150.205} C_DIS
LIN {X -0.053,Y -396.754,Z 661.619,A 0.000,B 0.000,C 90.000,E1 147.375} C_DIS
LIN {X -0.051,Y -397.559,Z 661.607,A 0.000,B 0.000,C 90.000,E1 145.261} C_DIS
LIN {X 0.096,Y -398.559,Z 661.595,A 0.000,B 0.000,C 90.000,E1 143.130} C_DIS
LIN {X -0.054,Y -399.651,Z 661.584,A 0.000,B 0.000,C 90.000,E1 141.045} C_DIS
LIN {X 0.014,Y -400.928,Z 661.572,A 0.000,B 0.000,C 90.000,E1 138.933} C_DIS
LIN {X -0.008,Y -401.951,Z 661.562,A 0.000,B 0.000,C 90.000,E1 137.187} C_DIS
LIN {X 0.072,Y -403.280,Z 661.551,A 0.000,B 0.000,C 90.000,E1 135.081} C_DIS
LIN {X -0.090,Y -404.888,Z 661.539,A 0.000,B 0.000,C 90.000,E1 133.014} C_DIS
LIN {X -0.258,Y -405.217,Z 661.537,A 0.000,B 0.000,C 90.000,E1 132.690} C_DIS
LIN {X -0.023,Y -406.374,Z 661.533,A 0.000,B 0.000,C 90.000,E1 131.962} C_DIS
LIN {X 0.112,Y -406.856,Z 661.531,A 0.000,B 0.000,C 90.000,E1 131.595} C_DIS
LIN {X -0.054,Y -407.937,Z 661.529,A 0.000,B 0.000,C 90.000,E1 131.272} C_DIS
LIN {X 0.090,Y -409.136,Z 661.527,A 0.000,B 0.000,C 90.000,E1 130.906} C_DIS
LIN {X 0.242,Y -410.981,Z 661.525,A 0.000,B 0.000,C 90.000,E1 130.539} C_DIS
LIN {X 0.165,Y -412.254,Z 661.524,A 0.000,B 0.000,C 90.000,E1 130.378} C_DIS
LIN {X -0.196,Y -415.184,Z 661.523,A 0.000,B 0.000,C 90.000,E1 130.092} C_DIS
LIN {X 0.161,Y -424.007,Z 661.518,A 0.000,B 0.000,C 90.000,E1 129.277} C_DIS
LIN {X -0.057,Y -448.024,Z 661.508,A 0.000,B 0.000,C 90.000,E1 127.523} C_DIS
LIN {X 0.087,Y -458.966,Z 661.504,A 0.000,B 0.000,C 90.000,E1 126.710} C_DIS
LIN {X 0.095,Y -465.214,Z 661.502,A 0.000,B 0.000,C 90.000,E1 126.251} C_DIS
LIN {X -0.067,Y -472.979,Z 661.498,A 0.000,B 0.000,C 90.000,E1 125.678} C_DIS
LIN {X -0.192,Y -480.315,Z 661.495,A 0.000,B 0.000,C 90.000,E1 125.105} C_DIS
LIN {X -0.214,Y -486.251,Z 661.492,A 0.000,B 0.000,C 90.000,E1 124.612} C_DIS
LIN {X 0.074,Y -490.632,Z 661.490,A 0.000,B 0.000,C 90.000,E1 124.199} C_DIS
LIN {X 0.124,Y -499.323,Z 661.486,A 0.000,B 0.000,C 90.000,E1 123.420} C_DIS
LIN {X 0.252,Y -510.430,Z 661.480,A 0.000,B 0.000,C 90.000,E1 122.339} C_DIS
LIN {X -0.117,Y -515.521,Z 661.477,A 0.000,B 0.000,C 90.000,E1 121.878} C_DIS
LIN {X -0.133,Y -523.531,Z 661.472,A 0.000,B 0.000,C 90.000,E1 121.052} C_DIS
LIN {X 0.117,Y -528.582,Z 661.469,A 0.000,B 0.000,C 90.000,E1 120.463} C_DIS
LIN {X -0.080,Y -532.214,Z 661.467,A 0.000,B 0.000,C 90.000,E1 120.050} C_DIS
LIN {X -0.086,Y -537.594,Z 661.463,A 0.000,B 0.000,C 90.000,E1 119.333} C_DIS
LIN {X 0.094,Y -541.583,Z 661.460,A 0.000,B 0.000,C 90.000,E1 118.743} C_DIS
LIN {X 0.177,Y -545.948,Z 661.456,A 0.000,B 0.000,C 90.000,E1 118.025} C_DIS
LIN {X 0.044,Y -549.880,Z 661.452,A 0.000,B 0.000,C 90.000,E1 117.334} C_DIS
LIN {X 0.204,Y -553.416,Z 661.448,A 0.000,B 0.000,C 90.000,E1 116.616} C_DIS
LIN {X 0.146,Y -556.718,Z 661.444,A 0.000,B 0.000,C 90.000,E1 115.924} C_DIS
LIN {X 0.252,Y -560.211,Z 661.440,A 0.000,B 0.000,C 90.000,E1 115.079} C_DIS
LIN {X -0.049,Y -564.486,Z 661.433,A 0.000,B 0.000,C 90.000,E1 114.003} C_DIS
LIN {X -0.001,Y -568.300,Z 661.427,A 0.000,B 0.000,C 90.000,E1 112.898} C_DIS
LIN {X -0.024,Y -570.890,Z 661.423,A 0.000,B 0.000,C 90.000,E1 112.078} C_DIS
LIN {X -0.063,Y -572.477,Z 661.420,A 0.000,B 0.000,C 90.000,E1 111.535} C_DIS
LIN {X -0.256,Y -574.607,Z 661.415,A 0.000,B 0.000,C 90.000,E1 110.737} C_DIS
LIN {X 0.113,Y -576.516,Z 661.411,A 0.000,B 0.000,C 90.000,E1 109.885} C_DIS
LIN {X -0.018,Y -579.498,Z 661.403,A 0.000,B 0.000,C 90.000,E1 108.544} C_DIS
LIN {X -0.285,Y -582.266,Z 661.396,A 0.000,B 0.000,C 90.000,E1 107.221} C_DIS
LIN {X 0.050,Y -585.116,Z 661.388,A 0.000,B 0.000,C 90.000,E1 105.843} C_DIS
LIN {X -0.289,Y -587.860,Z 661.381,A 0.000,B 0.000,C 90.000,E1 104.537} C_DIS
LIN {X -0.017,Y -590.560,Z 661.373,A 0.000,B 0.000,C 90.000,E1 103.175} C_DIS
LIN {X -0.107,Y -592.681,Z 661.367,A 0.000,B 0.000,C 90.000,E1 102.119} C_DIS
LIN {X -0.020,Y -596.360,Z 661.357,A 0.000,B 0.000,C 90.000,E1 100.254} C_DIS
LIN {X 0.062,Y -599.872,Z 661.347,A 0.000,B 0.000,C 90.000,E1 98.398} C_DIS
LIN {X 0.211,Y -602.118,Z 661.339,A 0.000,B 0.000,C 90.000,E1 97.068} C_DIS
LIN {X 0.091,Y -603.837,Z 661.334,A 0.000,B 0.000,C 90.000,E1 96.030} C_DIS
LIN {X 0.204,Y -606.537,Z 661.323,A 0.000,B 0.000,C 90.000,E1 94.188} C_DIS
LIN {X -0.214,Y -608.144,Z 661.316,A 0.000,B 0.000,C 90.000,E1 92.922} C_DIS
LIN {X 0.273,Y -609.323,Z 661.310,A 0.000,B 0.000,C 90.000,E1 91.835} C_DIS
LIN {X -0.138,Y -610.425,Z 661.303,A 0.000,B 0.000,C 90.000,E1 90.573} C_DIS
LIN {X 0.105,Y -610.944,Z 661.299,A 0.000,B 0.000,C 90.000,E1 89.771} C_DIS
LIN {X -0.299,Y -611.569,Z 661.292,A 0.000,B 0.000,C 90.000,E1 88.511} C_DIS
LIN {X 0.258,Y -611.855,Z 661.286,A 0.000,B 0.000,C 90.000,E1 87.421} C_DIS
LIN {X 0.212,Y -612.028,Z 661.280,A 0.000,B 0.000,C 90.000,E1 86.388} C_DIS
LIN {X 0.164,Y -611.969,Z 661.274,A 0.000,B 0.000,C 90.000,E1 85.355} C_DIS
LIN {X 0.165,Y -611.756,Z 661.269,A 0.000,B 0.000,C 90.000,E1 84.318} C_DIS
LIN {X -0.173,Y -611.206,Z 661.261,A 0.000,B 0.000,C 90.000,E1 83.053} C_DIS
LIN {X -0.102,Y -610.662,Z 661.256,A 0.000,B 0.000,C 90.000,E1 82.008} C_DIS
LIN {X 0.231,Y -610.037,Z 661.251,A 0.000,B 0.000,C 90.000,E1 81.197} C_DIS
LIN {X 0.295,Y -609.015,Z 661.245,A 0.000,B 0.000,C 90.000,E1 80.151} C_DIS
LIN {X 0.079,Y -607.500,Z 661.238,A 0.000,B 0.000,C 90.000,E1 78.870} C_DIS
LIN {X -0.170,Y -605.786,Z 661.231,A 0.000,B 0.000,C 90.000,E1 77.589} C_DIS
LIN {X 0.084,Y -604.267,Z 661.225,A 0.000,B 0.000,C 90.000,E1 76.520} C_DIS
LIN {X -0.094,Y -602.214,Z 661.218,A 0.000,B 0.000,C 90.000,E1 75.227} C_DIS
LIN {X 0.119,Y -600.457,Z 661.212,A 0.000,B 0.000,C 90.000,E1 74.157} C_DIS
LIN {X -0.269,Y -598.566,Z 661.206,A 0.000,B 0.000,C 90.000,E1 73.142} C_DIS
LIN {X -0.227,Y -596.047,Z 661.199,A 0.000,B 0.000,C 90.000,E1 71.819} C_DIS
LIN {X 0.186,Y -594.440,Z 661.195,A 0.000,B 0.000,C 90.000,E1 70.986} C_DIS
LIN {X 0.098,Y -592.163,Z 661.189,A 0.000,B 0.000,C 90.000,E1 69.934} C_DIS
LIN {X -0.217,Y -589.483,Z 661.183,A 0.000,B 0.000,C 90.000,E1 68.901} C_DIS
LIN {X 0.098,Y -588.100,Z 661.180,A 0.000,B 0.000,C 90.000,E1 68.337} C_DIS
LIN {X 0.065,Y -585.771,Z 661.175,A 0.000,B 0.000,C 90.000,E1 67.539} C_DIS
LIN {X 0.130,Y -584.119,Z 661.172,A 0.000,B 0.000,C 90.000,E1 66.997} C_DIS
LIN {X -0.257,Y -581.439,Z 661.168,A 0.000,B 0.000,C 90.000,E1 66.230} C_DIS
LIN {X -0.131,Y -578.507,Z 661.163,A 0.000,B 0.000,C 90.000,E1 65.409} C_DIS
LIN {X -0.037,Y -575.449,Z 661.159,A 0.000,B 0.000,C 90.000,E1 64.588} C_DIS
LIN {X -0.137,Y -571.029,Z 661.153,A 0.000,B 0.000,C 90.000,E1 63.512} C_DIS
LIN {X -0.045,Y -568.040,Z 661.149,A 0.000,B 0.000,C 90.000,E1 62.820} C_DIS
LIN {X -0.223,Y -564.933,Z 661.145,A 0.000,B 0.000,C 90.000,E1 62.153} C_DIS
LIN {X 0.069,Y -561.458,Z 661.141,A 0.000,B 0.000,C 90.000,E1 61.435} C_DIS
LIN {X 0.056,Y -557.539,Z 661.138,A 0.000,B 0.000,C 90.000,E1 60.745} C_DIS
LIN {X -0.098,Y -554.095,Z 661.134,A 0.000,B 0.000,C 90.000,E1 60.205} C_DIS
LIN {X 0.085,Y -549.298,Z 661.131,A 0.000,B 0.000,C 90.000,E1 59.488} C_DIS
LIN {X -0.190,Y -545.458,Z 661.128,A 0.000,B 0.000,C 90.000,E1 58.997} C_DIS
LIN {X 0.045,Y -540.690,Z 661.125,A 0.000,B 0.000,C 90.000,E1 58.408} C_DIS
LIN {X -0.128,Y -535.465,Z 661.121,A 0.000,B 0.000,C 90.000,E1 57.867} C_DIS
LIN {X 0.049,Y -531.214,Z 661.119,A 0.000,B 0.000,C 90.000,E1 57.454} C_DIS
LIN {X 0.069,Y -525.718,Z 661.117,A 0.000,B 0.000,C 90.000,E1 56.993} C_DIS
LIN {X -0.121,Y -519.918,Z 661.114,A 0.000,B 0.000,C 90.000,E1 56.580} C_DIS
LIN {X -0.085,Y -513.183,Z 661.112,A 0.000,B 0.000,C 90.000,E1 56.135} C_DIS
LIN {X 0.059,Y -506.464,Z 661.110,A 0.000,B 0.000,C 90.000,E1 55.722} C_DIS
LIN {X -0.229,Y -499.998,Z 661.108,A 0.000,B 0.000,C 90.000,E1 55.388} C_DIS
LIN {X 0.159,Y -480.075,Z 661.102,A 0.000,B 0.000,C 90.000,E1 54.276} C_DIS
LIN {X 0.041,Y -461.595,Z 661.096,A 0.000,B 0.000,C 90.000,E1 53.290} C_DIS
LIN {X 0.173,Y -433.060,Z 661.087,A 0.000,B 0.000,C 90.000,E1 51.618} C_DIS
LIN {X 0.129,Y -433.003,Z 661.087,A 0.000,B 0.000,C 90.000,E1 51.618} C_DIS
LIN {X 0.103,Y -431.512,Z 661.082,A 0.000,B 0.000,C 90.000,E1 50.803} C_DIS
LIN {X 0.011,Y -421.626,Z 661.058,A 0.000,B 0.000,C 90.000,E1 46.458} C_DIS
LIN {X 0.129,Y -418.842,Z 661.050,A 0.000,B 0.000,C 90.000,E1 44.919} C_DIS
LIN {X 0.073,Y -418.710,Z 661.049,A 0.000,B 0.000,C 90.000,E1 44.757} C_DIS
LIN {X -0.043,Y -418.827,Z 661.038,A 0.000,B 0.000,C 90.000,E1 42.894} C_DIS
LIN {X -0.095,Y -419.132,Z 661.027,A 0.000,B 0.000,C 90.000,E1 40.862} C_DIS
LIN {X 0.271,Y -419.902,Z 661.012,A 0.000,B 0.000,C 90.000,E1 38.096} C_DIS
LIN {X -0.165,Y -421.394,Z 660.995,A 0.000,B 0.000,C 90.000,E1 35.105} C_DIS
LIN {X 0.076,Y -422.606,Z 660.982,A 0.000,B 0.000,C 90.000,E1 32.704} C_DIS
LIN {X 0.195,Y -423.299,Z 660.974,A 0.000,B 0.000,C 90.000,E1 31.337} C_DIS
LIN {X 0.054,Y -424.370,Z 660.963,A 0.000,B 0.000,C 90.000,E1 29.333} C_DIS
LIN {X -0.103,Y -425.508,Z 660.952,A 0.000,B 0.000,C 90.000,E1 27.334} C_DIS
LIN {X -0.117,Y -428.043,Z 660.931,A 0.000,B 0.000,C 90.000,E1 23.643} C_DIS
LIN {X 0.036,Y -430.140,Z 660.918,A 0.000,B 0.000,C 90.000,E1 21.280} C_DIS
LIN {X -0.132,Y -431.058,Z 660.913,A 0.000,B 0.000,C 90.000,E1 20.301} C_DIS
LIN {X 0.151,Y -432.207,Z 660.904,A 0.000,B 0.000,C 90.000,E1 18.598} C_DIS
LIN {X -0.185,Y -433.727,Z 660.891,A 0.000,B 0.000,C 90.000,E1 16.315} C_DIS
LIN {X 0.127,Y -435.544,Z 660.878,A 0.000,B 0.000,C 90.000,E1 13.953} C_DIS
LIN {X -0.163,Y -437.310,Z 660.867,A 0.000,B 0.000,C 90.000,E1 12.007} C_DIS
LIN {X 0.212,Y -439.938,Z 660.852,A 0.000,B 0.000,C 90.000,E1 9.321} C_DIS
LIN {X 0.023,Y -442.855,Z 660.837,A 0.000,B 0.000,C 90.000,E1 6.720} C_DIS
LIN {X 0.021,Y -445.217,Z 660.826,A 0.000,B 0.000,C 90.000,E1 4.759} C_DIS
LIN {X -0.003,Y -447.849,Z 660.816,A 0.000,B 0.000,C 90.000,E1 2.808} C_DIS
LIN {X 0.018,Y -450.557,Z 660.805,A 0.000,B 0.000,C 90.000,E1 0.859} C_DIS
LIN {X 0.127,Y -454.872,Z 660.790,A 0.000,B 0.000,C 90.000,E1 358.165} C_DIS
LIN {X -0.137,Y -458.140,Z 660.779,A 0.000,B 0.000,C 90.000,E1 356.274} C_DIS
LIN {X 0.189,Y -461.585,Z 660.769,A 0.000,B 0.000,C 90.000,E1 354.318} C_DIS
LIN {X 0.188,Y -465.056,Z 660.758,A 0.000,B 0.000,C 90.000,E1 352.413} C_DIS
LIN {X -0.210,Y -467.354,Z 660.751,A 0.000,B 0.000,C 90.000,E1 351.197} C_DIS
LIN {X 0.158,Y -470.147,Z 660.742,A 0.000,B 0.000,C 90.000,E1 349.577} C_DIS
LIN {X -0.173,Y -472.913,Z 660.734,A 0.000,B 0.000,C 90.000,E1 348.049} C_DIS
LIN {X -0.144,Y -476.277,Z 660.723,A 0.000,B 0.000,C 90.000,E1 346.172} C_DIS
LIN {X 0.068,Y -479.785,Z 660.713,A 0.000,B 0.000,C 90.000,E1 344.283} C_DIS
LIN {X 0.163,Y -483.343,Z 660.702,A 0.000,B 0.000,C 90.000,E1 342.417} C_DIS
LIN {X -0.096,Y -487.562,Z 660.690,A 0.000,B 0.000,C 90.000,E1 340.296} C_DIS
LIN {X -0.175,Y -490.036,Z 660.684,A 0.000,B 0.000,C 90.000,E1 339.082} C_DIS
LIN {X -0.006,Y -493.024,Z 660.675,A 0.000,B 0.000,C 90.000,E1 337.539} C_DIS
LIN {X 0.167,Y -495.312,Z 660.669,A 0.000,B 0.000,C 90.000,E1 336.305} C_DIS
LIN {X 0.117,Y -497.398,Z 660.662,A 0.000,B 0.000,C 90.000,E1 335.101} C_DIS
LIN {X -0.006,Y -500.547,Z 660.652,A 0.000,B 0.000,C 90.000,E1 333.307} C_DIS
LIN {X -0.125,Y -503.364,Z 660.643,A 0.000,B 0.000,C 90.000,E1 331.820} C_DIS
LIN {X 0.056,Y -505.241,Z 660.639,A 0.000,B 0.000,C 90.000,E1 331.051} C_DIS
LIN {X -0.273,Y -506.743,Z 660.637,A 0.000,B 0.000,C 90.000,E1 330.667} C_DIS
LIN {X -0.142,Y -508.200,Z 660.634,A 0.000,B 0.000,C 90.000,E1 330.205} C_DIS
LIN {X 0.108,Y -510.275,Z 660.632,A 0.000,B 0.000,C 90.000,E1 329.793} C_DIS
LIN {X 0.236,Y -511.914,Z 660.631,A 0.000,B 0.000,C 90.000,E1 329.537} C_DIS
LIN {X -0.064,Y -517.250,Z 660.628,A 0.000,B 0.000,C 90.000,E1 328.997} C_DIS
LIN {X -0.129,Y -524.012,Z 660.625,A 0.000,B 0.000,C 90.000,E1 328.456} C_DIS
LIN {X 0.029,Y -534.361,Z 660.620,A 0.000,B 0.000,C 90.000,E1 327.661} C_DIS
LIN {X 0.093,Y -543.286,Z 660.617,A 0.000,B 0.000,C 90.000,E1 326.962} C_DIS
LIN {X 0.196,Y -554.458,Z 660.611,A 0.000,B 0.000,C 90.000,E1 326.008} C_DIS
LIN {X -0.209,Y -562.750,Z 660.607,A 0.000,B 0.000,C 90.000,E1 325.308} C_DIS
LIN {X 0.030,Y -573.416,Z 660.602,A 0.000,B 0.000,C 90.000,E1 324.276} C_DIS
LIN {X -0.112,Y -582.495,Z 660.597,A 0.000,B 0.000,C 90.000,E1 323.417} C_DIS
LIN {X -0.247,Y -587.626,Z 660.594,A 0.000,B 0.000,C 90.000,E1 322.924} C_DIS
LIN {X -0.254,Y -597.708,Z 660.588,A 0.000,B 0.000,C 90.000,E1 321.904} C_DIS
LIN {X -0.126,Y -602.679,Z 660.585,A 0.000,B 0.000,C 90.000,E1 321.376} C_DIS
LIN {X -0.043,Y -607.385,Z 660.583,A 0.000,B 0.000,C 90.000,E1 320.848} C_DIS
LIN {X -0.025,Y -612.987,Z 660.579,A 0.000,B 0.000,C 90.000,E1 320.194} C_DIS
LIN {X 0.039,Y -618.262,Z 660.575,A 0.000,B 0.000,C 90.000,E1 319.542} C_DIS
LIN {X 0.035,Y -623.974,Z 660.571,A 0.000,B 0.000,C 90.000,E1 318.771} C_DIS
LIN {X -0.288,Y -628.475,Z 660.567,A 0.000,B 0.000,C 90.000,E1 318.162} C_DIS
LIN {X 0.204,Y -634.477,Z 660.563,A 0.000,B 0.000,C 90.000,E1 317.229} C_DIS
LIN {X -0.133,Y -640.062,Z 660.558,A 0.000,B 0.000,C 90.000,E1 316.377} C_DIS
LIN {X 0.009,Y -646.222,Z 660.552,A 0.000,B 0.000,C 90.000,E1 315.364} C_DIS
LIN {X 0.179,Y -653.521,Z 660.545,A 0.000,B 0.000,C 90.000,E1 314.109} C_DIS
LIN {X 0.056,Y -658.243,Z 660.540,A 0.000,B 0.000,C 90.000,E1 313.257} C_DIS
LIN {X 0.002,Y -660.835,Z 660.538,A 0.000,B 0.000,C 90.000,E1 312.771} C_DIS
LIN {X -0.049,Y -666.357,Z 660.532,A 0.000,B 0.000,C 90.000,E1 311.676} C_DIS
LIN {X -0.004,Y -670.983,Z 660.526,A 0.000,B 0.000,C 90.000,E1 310.701} C_DIS
LIN {X 0.106,Y -675.177,Z 660.521,A 0.000,B 0.000,C 90.000,E1 309.725} C_DIS
LIN {X 0.248,Y -677.999,Z 660.517,A 0.000,B 0.000,C 90.000,E1 308.991} C_DIS
LIN {X 0.022,Y -681.373,Z 660.511,A 0.000,B 0.000,C 90.000,E1 308.051} C_DIS
LIN {X 0.227,Y -683.675,Z 660.507,A 0.000,B 0.000,C 90.000,E1 307.317} C_DIS
LIN {X 0.072,Y -686.566,Z 660.502,A 0.000,B 0.000,C 90.000,E1 306.377} C_DIS
LIN {X -0.055,Y -689.121,Z 660.497,A 0.000,B 0.000,C 90.000,E1 305.438} C_DIS
LIN {X 0.014,Y -691.544,Z 660.492,A 0.000,B 0.000,C 90.000,E1 304.485} C_DIS
LIN {X -0.454,Y -693.745,Z 660.486,A 0.000,B 0.000,C 90.000,E1 303.579} C_DIS
LIN {X 0.296,Y -696.235,Z 660.480,A 0.000,B 0.000,C 90.000,E1 302.339} C_DIS
LIN {X 0.096,Y -698.002,Z 660.475,A 0.000,B 0.000,C 90.000,E1 301.416} C_DIS
LIN {X 0.284,Y -699.622,Z 660.469,A 0.000,B 0.000,C 90.000,E1 300.463} C_DIS
LIN {X -0.136,Y -700.668,Z 660.466,A 0.000,B 0.000,C 90.000,E1 299.795} C_DIS
LIN {X -0.005,Y -702.147,Z 660.459,A 0.000,B 0.000,C 90.000,E1 298.615} C_DIS
LIN {X -0.180,Y -703.446,Z 660.453,A 0.000,B 0.000,C 90.000,E1 297.462} C_DIS
LIN {X -0.014,Y -704.645,Z 660.446,A 0.000,B 0.000,C 90.000,E1 296.283} C_DIS
LIN {X -0.095,Y -704.906,Z 660.442,A 0.000,B 0.000,C 90.000,E1 295.591} C_DIS
LIN {X 0.181,Y -704.300,Z 660.440,A 0.000,B 0.000,C 90.000,E1 295.103} C_DIS
LIN {X -0.170,Y -703.846,Z 660.438,A 0.000,B 0.000,C 90.000,E1 294.899} C_DIS
LIN {X 0.114,Y -702.662,Z 660.437,A 0.000,B 0.000,C 90.000,E1 294.643} C_DIS
LIN {X -0.394,Y -700.529,Z 660.435,A 0.000,B 0.000,C 90.000,E1 294.335} C_DIS
LIN {X -0.257,Y -699.638,Z 660.434,A 0.000,B 0.000,C 90.000,E1 294.207} C_DIS
LIN {X -0.121,Y -698.309,Z 660.434,A 0.000,B 0.000,C 90.000,E1 294.079} C_DIS
LIN {X -0.179,Y -694.854,Z 660.433,A 0.000,B 0.000,C 90.000,E1 293.875} C_DIS
LIN {X -0.108,Y -691.631,Z 660.432,A 0.000,B 0.000,C 90.000,E1 293.695} C_DIS
LIN {X 0.157,Y -689.828,Z 660.431,A 0.000,B 0.000,C 90.000,E1 293.590} C_DIS
LIN {X -0.089,Y -683.333,Z 660.430,A 0.000,B 0.000,C 90.000,E1 293.462} C_DIS
LIN {X -0.096,Y -679.165,Z 660.430,A 0.000,B 0.000,C 90.000,E1 293.387} C_DIS
LIN {X 0.161,Y -670.000,Z 660.429,A 0.000,B 0.000,C 90.000,E1 293.259} C_DIS
LIN {X -0.116,Y -662.721,Z 660.429,A 0.000,B 0.000,C 90.000,E1 293.206} C_DIS
LIN {X -0.227,Y -652.784,Z 660.428,A 0.000,B 0.000,C 90.000,E1 293.078} C_DIS
LIN {X -0.139,Y -643.071,Z 660.427,A 0.000,B 0.000,C 90.000,E1 292.898} C_DIS
LIN {X 0.112,Y -629.558,Z 660.426,A 0.000,B 0.000,C 90.000,E1 292.589} C_DIS
LIN {X -0.256,Y -616.238,Z 660.424,A 0.000,B 0.000,C 90.000,E1 292.280} C_DIS
LIN {X 0.212,Y -588.949,Z 660.419,A 0.000,B 0.000,C 90.000,E1 291.408} C_DIS
LIN {X -0.028,Y -576.565,Z 660.417,A 0.000,B 0.000,C 90.000,E1 291.046} C_DIS
LIN {X 0.121,Y -564.245,Z 660.415,A 0.000,B 0.000,C 90.000,E1 290.684} C_DIS
LIN {X -0.156,Y -561.545,Z 660.414,A 0.000,B 0.000,C 90.000,E1 290.610} C_DIS
LIN {X 0.235,Y -556.267,Z 660.413,A 0.000,B 0.000,C 90.000,E1 290.301} C_DIS
LIN {X 0.188,Y -556.235,Z 660.413,A 0.000,B 0.000,C 90.000,E1 290.301} C_DIS
LIN {X -0.010,Y -555.446,Z 660.412,A 0.000,B 0.000,C 90.000,E1 290.174} C_DIS
LIN {X -0.101,Y -555.005,Z 660.410,A 0.000,B 0.000,C 90.000,E1 289.885} C_DIS
LIN {X -0.020,Y -554.686,Z 660.407,A 0.000,B 0.000,C 90.000,E1 289.322} C_DIS
LIN {X 0.228,Y -554.571,Z 660.401,A 0.000,B 0.000,C 90.000,E1 288.181} C_DIS
LIN {X 0.063,Y -554.224,Z 660.393,A 0.000,B 0.000,C 90.000,E1 286.804} C_DIS
LIN {X 0.306,Y -553.885,Z 660.387,A 0.000,B 0.000,C 90.000,E1 285.662} C_DIS
LIN {X -0.027,Y -553.290,Z 660.379,A 0.000,B 0.000,C 90.000,E1 284.300} C_DIS
LIN {X 0.285,Y -552.411,Z 660.370,A 0.000,B 0.000,C 90.000,E1 282.591} C_DIS
LIN {X 0.031,Y -551.393,Z 660.359,A 0.000,B 0.000,C 90.000,E1 280.658} C_DIS
LIN {X 0.104,Y -550.699,Z 660.348,A 0.000,B 0.000,C 90.000,E1 278.690} C_DIS
LIN {X -0.239,Y -550.056,Z 660.334,A 0.000,B 0.000,C 90.000,E1 276.201} C_DIS
LIN {X 0.228,Y -549.775,Z 660.323,A 0.000,B 0.000,C 90.000,E1 274.188} C_DIS
LIN {X -0.002,Y -549.526,Z 660.316,A 0.000,B 0.000,C 90.000,E1 272.808} C_DIS
LIN {X 0.155,Y -549.313,Z 660.311,A 0.000,B 0.000,C 90.000,E1 271.949} C_DIS
LIN {X -0.117,Y -548.733,Z 660.303,A 0.000,B 0.000,C 90.000,E1 270.573} C_DIS
LIN {X 0.136,Y -548.092,Z 660.295,A 0.000,B 0.000,C 90.000,E1 269.141} C_DIS
LIN {X -0.113,Y -547.127,Z 660.286,A 0.000,B 0.000,C 90.000,E1 267.478} C_DIS
LIN {X 0.120,Y -546.345,Z 660.278,A 0.000,B 0.000,C 90.000,E1 266.045} C_DIS
LIN {X -0.097,Y -545.034,Z 660.269,A 0.000,B 0.000,C 90.000,E1 264.375} C_DIS
LIN {X 0.107,Y -544.074,Z 660.262,A 0.000,B 0.000,C 90.000,E1 263.223} C_DIS
LIN {X -0.008,Y -542.011,Z 660.251,A 0.000,B 0.000,C 90.000,E1 261.254} C_DIS
LIN {X 0.031,Y -539.279,Z 660.236,A 0.000,B 0.000,C 90.000,E1 258.409} C_DIS
LIN {X 0.030,Y -537.797,Z 660.226,A 0.000,B 0.000,C 90.000,E1 256.700} C_DIS
LIN {X -0.112,Y -536.860,Z 660.220,A 0.000,B 0.000,C 90.000,E1 255.574} C_DIS
LIN {X 0.250,Y -535.887,Z 660.214,A 0.000,B 0.000,C 90.000,E1 254.393} C_DIS
LIN {X 0.073,Y -534.736,Z 660.207,A 0.000,B 0.000,C 90.000,E1 253.268} C_DIS
LIN {X -0.253,Y -533.072,Z 660.198,A 0.000,B 0.000,C 90.000,E1 251.583} C_DIS
LIN {X -0.146,Y -531.900,Z 660.191,A 0.000,B 0.000,C 90.000,E1 250.423} C_DIS
LIN {X -0.246,Y -530.876,Z 660.186,A 0.000,B 0.000,C 90.000,E1 249.571} C_DIS
LIN {X 0.197,Y -528.439,Z 660.177,A 0.000,B 0.000,C 90.000,E1 247.794} C_DIS
LIN {X 0.251,Y -527.176,Z 660.172,A 0.000,B 0.000,C 90.000,E1 246.922} C_DIS
LIN {X -0.020,Y -525.330,Z 660.166,A 0.000,B 0.000,C 90.000,E1 245.793} C_DIS
LIN {X 0.065,Y -522.701,Z 660.157,A 0.000,B 0.000,C 90.000,E1 244.332} C_DIS
LIN {X -0.041,Y -520.483,Z 660.151,A 0.000,B 0.000,C 90.000,E1 243.179} C_DIS
LIN {X -0.143,Y -516.896,Z 660.141,A 0.000,B 0.000,C 90.000,E1 241.435} C_DIS
LIN {X 0.007,Y -513.706,Z 660.133,A 0.000,B 0.000,C 90.000,E1 239.950} C_DIS
LIN {X 0.166,Y -510.380,Z 660.125,A 0.000,B 0.000,C 90.000,E1 238.456} C_DIS
LIN {X -0.107,Y -506.412,Z 660.115,A 0.000,B 0.000,C 90.000,E1 236.707} C_DIS
LIN {X 0.001,Y -504.286,Z 660.110,A 0.000,B 0.000,C 90.000,E1 235.801} C_DIS
LIN {X -0.142,Y -500.524,Z 660.102,A 0.000,B 0.000,C 90.000,E1 234.322} C_DIS
LIN {X 0.041,Y -496.634,Z 660.093,A 0.000,B 0.000,C 90.000,E1 232.798} C_DIS
LIN {X 0.047,Y -491.484,Z 660.082,A 0.000,B 0.000,C 90.000,E1 230.678} C_DIS
LIN {X 0.030,Y -487.202,Z 660.071,A 0.000,B 0.000,C 90.000,E1 228.852} C_DIS
LIN {X -0.081,Y -482.825,Z 660.061,A 0.000,B 0.000,C 90.000,E1 227.025} C_DIS
LIN {X -0.107,Y -479.195,Z 660.053,A 0.000,B 0.000,C 90.000,E1 225.486} C_DIS
LIN {X -0.210,Y -473.270,Z 660.039,A 0.000,B 0.000,C 90.000,E1 223.014} C_DIS
LIN {X 0.193,Y -467.647,Z 660.025,A 0.000,B 0.000,C 90.000,E1 220.458} C_DIS
LIN {X 0.005,Y -463.768,Z 660.014,A 0.000,B 0.000,C 90.000,E1 218.588} C_DIS
LIN {X 0.028,Y -461.124,Z 660.007,A 0.000,B 0.000,C 90.000,E1 217.317} C_DIS
LIN {X -0.125,Y -456.688,Z 659.995,A 0.000,B 0.000,C 90.000,E1 215.105} C_DIS
LIN {X -0.107,Y -453.700,Z 659.986,A 0.000,B 0.000,C 90.000,E1 213.499} C_DIS
LIN {X 0.069,Y -450.094,Z 659.975,A 0.000,B 0.000,C 90.000,E1 211.544} C_DIS
LIN {X -0.065,Y -446.536,Z 659.965,A 0.000,B 0.000,C 90.000,E1 209.617} C_DIS
LIN {X -0.054,Y -442.412,Z 659.952,A 0.000,B 0.000,C 90.000,E1 207.334} C_DIS
LIN {X 0.190,Y -438.920,Z 659.941,A 0.000,B 0.000,C 90.000,E1 205.335} C_DIS
LIN {X -0.034,Y -435.366,Z 659.930,A 0.000,B 0.000,C 90.000,E1 203.387} C_DIS
LIN {X -0.154,Y -432.921,Z 659.923,A 0.000,B 0.000,C 90.000,E1 202.078} C_DIS
LIN {X 0.147,Y -429.950,Z 659.913,A 0.000,B 0.000,C 90.000,E1 200.375} C_DIS
LIN {X 0.194,Y -426.441,Z 659.902,A 0.000,B 0.000,C 90.000,E1 198.362} C_DIS
LIN {X -0.108,Y -423.088,Z 659.891,A 0.000,B 0.000,C 90.000,E1 196.386} C_DIS
LIN {X -0.087,Y -419.787,Z 659.880,A 0.000,B 0.000,C 90.000,E1 194.356} C_DIS
LIN {X -0.006,Y -416.973,Z 659.870,A 0.000,B 0.000,C 90.000,E1 192.647} C_DIS
LIN {X 0.017,Y -413.275,Z 659.857,A 0.000,B 0.000,C 90.000,E1 190.254} C_DIS
LIN {X -0.196,Y -410.707,Z 659.847,A 0.000,B 0.000,C 90.000,E1 188.568} C_DIS
LIN {X -0.117,Y -408.145,Z 659.838,A 0.000,B 0.000,C 90.000,E1 186.834} C_DIS
LIN {X 0.203,Y -403.907,Z 659.821,A 0.000,B 0.000,C 90.000,E1 183.669} C_DIS
LIN {X -0.020,Y -401.048,Z 659.807,A 0.000,B 0.000,C 90.000,E1 181.260} C_DIS
LIN {X -0.083,Y -397.821,Z 659.788,A 0.000,B 0.000,C 90.000,E1 177.764} C_DIS
LIN {X -0.173,Y -395.820,Z 659.770,A 0.000,B 0.000,C 90.000,E1 174.609} C_DIS
LIN {X -0.153,Y -394.620,Z 659.754,A 0.000,B 0.000,C 90.000,E1 171.781} C_DIS
LIN {X 0.018,Y -393.960,Z 659.739,A 0.000,B 0.000,C 90.000,E1 168.926} C_DIS
LIN {X -0.093,Y -393.682,Z 659.725,A 0.000,B 0.000,C 90.000,E1 166.464} C_DIS
LIN {X -0.083,Y -393.714,Z 659.713,A 0.000,B 0.000,C 90.000,E1 164.338} C_DIS
LIN {X -0.061,Y -394.031,Z 659.695,A 0.000,B 0.000,C 90.000,E1 161.148} C_DIS
LIN {X -0.141,Y -394.327,Z 659.685,A 0.000,B 0.000,C 90.000,E1 159.390} C_DIS
LIN {X -0.191,Y -394.779,Z 659.672,A 0.000,B 0.000,C 90.000,E1 156.922} C_DIS
LIN {X -0.062,Y -395.342,Z 659.656,A 0.000,B 0.000,C 90.000,E1 154.076} C_DIS
LIN {X -0.183,Y -395.780,Z 659.644,A 0.000,B 0.000,C 90.000,E1 151.975} C_DIS
LIN {X -0.147,Y -396.238,Z 659.634,A 0.000,B 0.000,C 90.000,E1 150.205} C_DIS
LIN {X -0.076,Y -397.006,Z 659.619,A 0.000,B 0.000,C 90.000,E1 147.375} C_DIS
LIN {X 0.031,Y -397.948,Z 659.605,A 0.000,B 0.000,C 90.000,E1 144.895} C_DIS
LIN {X 0.085,Y -398.797,Z 659.595,A 0.000,B 0.000,C 90.000,E1 143.130} C_DIS
LIN {X 0.079,Y -399.676,Z 659.586,A 0.000,B 0.000,C 90.000,E1 141.376} C_DIS
LIN {X 0.013,Y -401.081,Z 659.572,A 0.000,B 0.000,C 90.000,E1 138.933} C_DIS
LIN {X -0.122,Y -401.908,Z 659.564,A 0.000,B 0.000,C 90.000,E1 137.553} C_DIS
LIN {X 0.077,Y -403.307,Z 659.551,A 0.000,B 0.000,C 90.000,E1 135.081} C_DIS
LIN {X -0.252,Y -405.187,Z 659.537,A 0.000,B 0.000,C 90.000,E1 132.690} C_DIS
LIN {X 0.118,Y -406.591,Z 659.531,A 0.000,B 0.000,C 90.000,E1 131.595} C_DIS
LIN {X 0.035,Y -406.910,Z 659.530,A 0.000,B 0.000,C 90.000,E1 131.434} C_DIS
LIN {X -0.050,Y -407.519,Z 659.529,A 0.000,B 0.000,C 90.000,E1 131.272} C_DIS
LIN {X 0.011,Y -408.990,Z 659.526,A 0.000,B 0.000,C 90.000,E1 130.744} C_DIS
LIN {X 0.160,Y -410.771,Z 659.524,A 0.000,B 0.000,C 90.000,E1 130.378} C_DIS
LIN {X -0.186,Y -411.850,Z 659.524,A 0.000,B 0.000,C 90.000,E1 130.253} C_DIS
LIN {X 0.011,Y -414.778,Z 659.522,A 0.000,B 0.000,C 90.000,E1 129.886} C_DIS
LIN {X 0.086,Y -424.119,Z 659.517,A 0.000,B 0.000,C 90.000,E1 129.072} C_DIS
LIN {X -0.150,Y -447.861,Z 659.508,A 0.000,B 0.000,C 90.000,E1 127.363} C_DIS
LIN {X 0.113,Y -462.314,Z 659.502,A 0.000,B 0.000,C 90.000,E1 126.297} C_DIS
LIN {X -0.211,Y -474.697,Z 659.497,A 0.000,B 0.000,C 90.000,E1 125.391} C_DIS
LIN {X 0.205,Y -482.267,Z 659.493,A 0.000,B 0.000,C 90.000,E1 124.739} C_DIS
LIN {X 0.159,Y -489.678,Z 659.490,A 0.000,B 0.000,C 90.000,E1 124.119} C_DIS
LIN {X -0.060,Y -498.443,Z 659.485,A 0.000,B 0.000,C 90.000,E1 123.372} C_DIS
LIN {X 0.064,Y -509.684,Z 659.479,A 0.000,B 0.000,C 90.000,E1 122.291} C_DIS
LIN {X 0.182,Y -513.839,Z 659.477,A 0.000,B 0.000,C 90.000,E1 121.878} C_DIS
LIN {X 0.172,Y -521.984,Z 659.473,A 0.000,B 0.000,C 90.000,E1 121.052} C_DIS
LIN {X -0.092,Y -528.109,Z 659.469,A 0.000,B 0.000,C 90.000,E1 120.413} C_DIS
LIN {X -0.153,Y -531.739,Z 659.467,A 0.000,B 0.000,C 90.000,E1 120.001} C_DIS
LIN {X -0.110,Y -537.222,Z 659.463,A 0.000,B 0.000,C 90.000,E1 119.283} C_DIS
LIN {X 0.069,Y -541.354,Z 659.459,A 0.000,B 0.000,C 90.000,E1 118.693} C_DIS
LIN {X -0.201,Y -545.040,Z 659.456,A 0.000,B 0.000,C 90.000,E1 118.153} C_DIS
LIN {X -0.091,Y -549.157,Z 659.452,A 0.000,B 0.000,C 90.000,E1 117.436} C_DIS
LIN {X -0.310,Y -553.468,Z 659.448,A 0.000,B 0.000,C 90.000,E1 116.616} C_DIS
LIN {X -0.126,Y -556.808,Z 659.444,A 0.000,B 0.000,C 90.000,E1 115.899} C_DIS
LIN {X -0.160,Y -559.766,Z 659.440,A 0.000,B 0.000,C 90.000,E1 115.207} C_DIS
LIN {X 0.048,Y -564.118,Z 659.434,A 0.000,B 0.000,C 90.000,E1 114.079} C_DIS
LIN {X -0.015,Y -567.115,Z 659.429,A 0.000,B 0.000,C 90.000,E1 113.259} C_DIS
LIN {X -0.269,Y -569.885,Z 659.425,A 0.000,B 0.000,C 90.000,E1 112.461} C_DIS
LIN {X 0.251,Y -572.369,Z 659.420,A 0.000,B 0.000,C 90.000,E1 111.589} C_DIS
LIN {X 0.054,Y -574.589,Z 659.416,A 0.000,B 0.000,C 90.000,E1 110.791} C_DIS
LIN {X 0.056,Y -577.152,Z 659.410,A 0.000,B 0.000,C 90.000,E1 109.704} C_DIS
LIN {X 0.288,Y -579.581,Z 659.404,A 0.000,B 0.000,C 90.000,E1 108.598} C_DIS
LIN {X 0.019,Y -582.379,Z 659.396,A 0.000,B 0.000,C 90.000,E1 107.275} C_DIS
LIN {X 0.026,Y -585.815,Z 659.387,A 0.000,B 0.000,C 90.000,E1 105.662} C_DIS
LIN {X 0.205,Y -589.719,Z 659.377,A 0.000,B 0.000,C 90.000,E1 103.772} C_DIS
LIN {X -0.197,Y -592.434,Z 659.369,A 0.000,B 0.000,C 90.000,E1 102.479} C_DIS
LIN {X 0.007,Y -596.123,Z 659.359,A 0.000,B 0.000,C 90.000,E1 100.602} C_DIS
LIN {X -0.120,Y -599.235,Z 659.350,A 0.000,B 0.000,C 90.000,E1 99.029} C_DIS
LIN {X -0.293,Y -601.179,Z 659.344,A 0.000,B 0.000,C 90.000,E1 97.992} C_DIS
LIN {X -0.123,Y -603.423,Z 659.337,A 0.000,B 0.000,C 90.000,E1 96.663} C_DIS
LIN {X -0.229,Y -605.071,Z 659.331,A 0.000,B 0.000,C 90.000,E1 95.625} C_DIS
LIN {X -0.059,Y -607.023,Z 659.324,A 0.000,B 0.000,C 90.000,E1 94.302} C_DIS
LIN {X 0.136,Y -608.729,Z 659.317,A 0.000,B 0.000,C 90.000,E1 92.980} C_DIS
LIN {X -0.288,Y -610.149,Z 659.309,A 0.000,B 0.000,C 90.000,E1 91.718} C_DIS
LIN {X -0.094,Y -611.239,Z 659.302,A 0.000,B 0.000,C 90.000,E1 90.401} C_DIS
LIN {X 0.157,Y -611.726,Z 659.298,A 0.000,B 0.000,C 90.000,E1 89.599} C_DIS
LIN {X 0.089,Y -612.226,Z 659.292,A 0.000,B 0.000,C 90.000,E1 88.568} C_DIS
LIN {X 0.044,Y -612.540,Z 659.286,A 0.000,B 0.000,C 90.000,E1 87.535} C_DIS
LIN {X 0.008,Y -612.715,Z 659.281,A 0.000,B 0.000,C 90.000,E1 86.502} C_DIS
LIN {X -0.029,Y -612.653,Z 659.275,A 0.000,B 0.000,C 90.000,E1 85.469} C_DIS
LIN {X 0.259,Y -612.319,Z 659.268,A 0.000,B 0.000,C 90.000,E1 84.147} C_DIS
LIN {X 0.001,Y -611.740,Z 659.260,A 0.000,B 0.000,C 90.000,E1 82.875} C_DIS
LIN {X 0.000,Y -611.123,Z 659.255,A 0.000,B 0.000,C 90.000,E1 81.837} C_DIS
LIN {X -0.268,Y -610.430,Z 659.250,A 0.000,B 0.000,C 90.000,E1 81.084} C_DIS
LIN {X -0.202,Y -609.361,Z 659.245,A 0.000,B 0.000,C 90.000,E1 80.038} C_DIS
LIN {X 0.181,Y -607.799,Z 659.237,A 0.000,B 0.000,C 90.000,E1 78.701} C_DIS
LIN {X 0.059,Y -606.016,Z 659.230,A 0.000,B 0.000,C 90.000,E1 77.409} C_DIS
LIN {X 0.178,Y -604.458,Z 659.224,A 0.000,B 0.000,C 90.000,E1 76.353} C_DIS
LIN {X 0.146,Y -602.350,Z 659.217,A 0.000,B 0.000,C 90.000,E1 75.046} C_DIS
LIN {X -0.215,Y -600.538,Z 659.211,A 0.000,B 0.000,C 90.000,E1 74.031} C_DIS
LIN {X -0.023,Y -598.583,Z 659.205,A 0.000,B 0.000,C 90.000,E1 72.960} C_DIS
LIN {X 0.017,Y -596.007,Z 659.198,A 0.000,B 0.000,C 90.000,E1 71.638} C_DIS
LIN {X -0.133,Y -594.334,Z 659.194,A 0.000,B 0.000,C 90.000,E1 70.859} C_DIS
LIN {X -0.106,Y -592.589,Z 659.189,A 0.000,B 0.000,C 90.000,E1 70.061} C_DIS
LIN {X 0.133,Y -589.886,Z 659.183,A 0.000,B 0.000,C 90.000,E1 68.975} C_DIS
LIN {X 0.330,Y -587.686,Z 659.179,A 0.000,B 0.000,C 90.000,E1 68.156} C_DIS
LIN {X 0.166,Y -584.468,Z 659.173,A 0.000,B 0.000,C 90.000,E1 67.102} C_DIS
LIN {X 0.087,Y -581.740,Z 659.168,A 0.000,B 0.000,C 90.000,E1 66.305} C_DIS
LIN {X 0.069,Y -577.733,Z 659.162,A 0.000,B 0.000,C 90.000,E1 65.229} C_DIS
LIN {X 0.152,Y -574.579,Z 659.158,A 0.000,B 0.000,C 90.000,E1 64.409} C_DIS
LIN {X 0.197,Y -571.237,Z 659.153,A 0.000,B 0.000,C 90.000,E1 63.589} C_DIS
LIN {X -0.045,Y -567.557,Z 659.149,A 0.000,B 0.000,C 90.000,E1 62.794} C_DIS
LIN {X 0.101,Y -565.051,Z 659.146,A 0.000,B 0.000,C 90.000,E1 62.231} C_DIS
LIN {X -0.082,Y -561.511,Z 659.142,A 0.000,B 0.000,C 90.000,E1 61.563} C_DIS
LIN {X 0.180,Y -557.568,Z 659.138,A 0.000,B 0.000,C 90.000,E1 60.845} C_DIS
LIN {X -0.081,Y -553.099,Z 659.134,A 0.000,B 0.000,C 90.000,E1 60.177} C_DIS
LIN {X -0.061,Y -549.204,Z 659.131,A 0.000,B 0.000,C 90.000,E1 59.616} C_DIS
LIN {X -0.142,Y -545.916,Z 659.129,A 0.000,B 0.000,C 90.000,E1 59.203} C_DIS
LIN {X -0.266,Y -544.881,Z 659.128,A 0.000,B 0.000,C 90.000,E1 59.076} C_DIS
LIN {X 0.246,Y -540.002,Z 659.125,A 0.000,B 0.000,C 90.000,E1 58.456} C_DIS
LIN {X 0.203,Y -534.731,Z 659.122,A 0.000,B 0.000,C 90.000,E1 57.916} C_DIS
LIN {X 0.139,Y -530.462,Z 659.120,A 0.000,B 0.000,C 90.000,E1 57.533} C_DIS
LIN {X -0.076,Y -524.683,Z 659.117,A 0.000,B 0.000,C 90.000,E1 57.089} C_DIS
LIN {X 0.202,Y -519.814,Z 659.115,A 0.000,B 0.000,C 90.000,E1 56.707} C_DIS
LIN {X 0.085,Y -513.299,Z 659.113,A 0.000,B 0.000,C 90.000,E1 56.294} C_DIS
LIN {X 0.149,Y -505.004,Z 659.110,A 0.000,B 0.000,C 90.000,E1 55.801} C_DIS
LIN {X -0.171,Y -498.303,Z 659.108,A 0.000,B 0.000,C 90.000,E1 55.468} C_DIS
LIN {X -0.130,Y -478.369,Z 659.102,A 0.000,B 0.000,C 90.000,E1 54.402} C_DIS
LIN {X -0.116,Y -461.569,Z 659.097,A 0.000,B 0.000,C 90.000,E1 53.497} C_DIS
LIN {X -0.173,Y -435.054,Z 659.089,A 0.000,B 0.000,C 90.000,E1 51.984} C_DIS
LIN {X 0.268,Y -433.460,Z 659.088,A 0.000,B 0.000,C 90.000,E1 51.823} C_DIS
LIN {X 0.245,Y -433.422,Z 659.088,A 0.000,B 0.000,C 90.000,E1 51.823} C_DIS
LIN {X -0.281,Y -431.400,Z 659.082,A 0.000,B 0.000,C 90.000,E1 50.803} C_DIS
LIN {X 0.020,Y -422.187,Z 659.060,A 0.000,B 0.000,C 90.000,E1 46.743} C_DIS
LIN {X -0.144,Y -419.341,Z 659.051,A 0.000,B 0.000,C 90.000,E1 45.243} C_DIS
LIN {X -0.198,Y -419.175,Z 659.050,A 0.000,B 0.000,C 90.000,E1 45.081} C_DIS
LIN {X -0.132,Y -419.311,Z 659.042,A 0.000,B 0.000,C 90.000,E1 43.542} C_DIS
LIN {X -0.008,Y -419.595,Z 659.029,A 0.000,B 0.000,C 90.000,E1 41.148} C_DIS
LIN {X -0.222,Y -420.353,Z 659.014,A 0.000,B 0.000,C 90.000,E1 38.463} C_DIS
LIN {X -0.053,Y -421.808,Z 658.997,A 0.000,B 0.000,C 90.000,E1 35.391} C_DIS
LIN {X -0.092,Y -422.639,Z 658.987,A 0.000,B 0.000,C 90.000,E1 33.706} C_DIS
LIN {X -0.001,Y -423.540,Z 658.978,A 0.000,B 0.000,C 90.000,E1 32.005} C_DIS
LIN {X -0.156,Y -424.761,Z 658.965,A 0.000,B 0.000,C 90.000,E1 29.667} C_DIS
LIN {X -0.105,Y -425.863,Z 658.954,A 0.000,B 0.000,C 90.000,E1 27.641} C_DIS
LIN {X -0.053,Y -427.234,Z 658.940,A 0.000,B 0.000,C 90.000,E1 25.283} C_DIS
LIN {X 0.052,Y -428.809,Z 658.929,A 0.000,B 0.000,C 90.000,E1 23.259} C_DIS
LIN {X -0.148,Y -430.615,Z 658.918,A 0.000,B 0.000,C 90.000,E1 21.280} C_DIS
LIN {X 0.095,Y -431.497,Z 658.913,A 0.000,B 0.000,C 90.000,E1 20.248} C_DIS
LIN {X -0.019,Y -432.635,Z 658.903,A 0.000,B 0.000,C 90.000,E1 18.598} C_DIS
LIN {X 0.074,Y -434.110,Z 658.890,A 0.000,B 0.000,C 90.000,E1 16.260} C_DIS
LIN {X 0.084,Y -435.908,Z 658.878,A 0.000,B 0.000,C 90.000,E1 13.939} C_DIS
LIN {X 0.125,Y -437.653,Z 658.867,A 0.000,B 0.000,C 90.000,E1 11.951} C_DIS
LIN {X 0.080,Y -440.261,Z 658.852,A 0.000,B 0.000,C 90.000,E1 9.321} C_DIS
LIN {X -0.099,Y -443.141,Z 658.837,A 0.000,B 0.000,C 90.000,E1 6.720} C_DIS
LIN {X -0.095,Y -445.483,Z 658.826,A 0.000,B 0.000,C 90.000,E1 4.759} C_DIS
LIN {X -0.114,Y -448.081,Z 658.816,A 0.000,B 0.000,C 90.000,E1 2.808} C_DIS
LIN {X -0.088,Y -450.772,Z 658.805,A 0.000,B 0.000,C 90.000,E1 0.859} C_DIS
LIN {X 0.131,Y -455.030,Z 658.790,A 0.000,B 0.000,C 90.000,E1 358.165} C_DIS
LIN {X 0.144,Y -457.718,Z 658.781,A 0.000,B 0.000,C 90.000,E1 356.560} C_DIS
LIN {X 0.199,Y -461.697,Z 658.769,A 0.000,B 0.000,C 90.000,E1 354.318} C_DIS
LIN {X 0.200,Y -465.152,Z 658.758,A 0.000,B 0.000,C 90.000,E1 352.413} C_DIS
LIN {X -0.196,Y -467.451,Z 658.751,A 0.000,B 0.000,C 90.000,E1 351.197} C_DIS
LIN {X 0.175,Y -470.243,Z 658.742,A 0.000,B 0.000,C 90.000,E1 349.577} C_DIS
LIN {X 0.137,Y -473.552,Z 658.732,A 0.000,B 0.000,C 90.000,E1 347.701} C_DIS
LIN {X 0.133,Y -477.510,Z 658.720,A 0.000,B 0.000,C 90.000,E1 345.519} C_DIS
LIN {X -0.089,Y -481.031,Z 658.709,A 0.000,B 0.000,C 90.000,E1 343.685} C_DIS
LIN {X 0.037,Y -484.034,Z 658.701,A 0.000,B 0.000,C 90.000,E1 342.127} C_DIS
LIN {X -0.217,Y -488.240,Z 658.689,A 0.000,B 0.000,C 90.000,E1 340.007} C_DIS
LIN {X -0.118,Y -490.713,Z 658.682,A 0.000,B 0.000,C 90.000,E1 338.773} C_DIS
LIN {X 0.064,Y -493.669,Z 658.674,A 0.000,B 0.000,C 90.000,E1 337.230} C_DIS
LIN {X -0.210,Y -495.881,Z 658.667,A 0.000,B 0.000,C 90.000,E1 336.049} C_DIS
LIN {X -0.196,Y -498.429,Z 658.658,A 0.000,B 0.000,C 90.000,E1 334.537} C_DIS
LIN {X 0.025,Y -500.513,Z 658.652,A 0.000,B 0.000,C 90.000,E1 333.307} C_DIS
LIN {X -0.031,Y -503.880,Z 658.642,A 0.000,B 0.000,C 90.000,E1 331.513} C_DIS
LIN {X -0.104,Y -505.356,Z 658.638,A 0.000,B 0.000,C 90.000,E1 330.923} C_DIS
LIN {X -0.160,Y -506.105,Z 658.637,A 0.000,B 0.000,C 90.000,E1 330.717} C_DIS
LIN {X -0.030,Y -507.334,Z 658.635,A 0.000,B 0.000,C 90.000,E1 330.255} C_DIS
LIN {X 0.109,Y -509.182,Z 658.632,A 0.000,B 0.000,C 90.000,E1 329.793} C_DIS
LIN {X -0.259,Y -510.755,Z 658.631,A 0.000,B 0.000,C 90.000,E1 329.537} C_DIS
LIN {X 0.077,Y -512.771,Z 658.629,A 0.000,B 0.000,C 90.000,E1 329.203} C_DIS
LIN {X -0.098,Y -515.897,Z 658.627,A 0.000,B 0.000,C 90.000,E1 328.869} C_DIS
LIN {X -0.074,Y -520.281,Z 658.625,A 0.000,B 0.000,C 90.000,E1 328.456} C_DIS
LIN {X -0.260,Y -533.597,Z 658.619,A 0.000,B 0.000,C 90.000,E1 327.454} C_DIS
LIN {X -0.089,Y -542.395,Z 658.615,A 0.000,B 0.000,C 90.000,E1 326.755} C_DIS
LIN {X -0.132,Y -552.367,Z 658.611,A 0.000,B 0.000,C 90.000,E1 325.928} C_DIS
LIN {X -0.036,Y -559.297,Z 658.607,A 0.000,B 0.000,C 90.000,E1 325.308} C_DIS
LIN {X -0.038,Y -567.457,Z 658.603,A 0.000,B 0.000,C 90.000,E1 324.562} C_DIS
LIN {X -0.268,Y -576.790,Z 658.598,A 0.000,B 0.000,C 90.000,E1 323.703} C_DIS
LIN {X -0.097,Y -584.674,Z 658.594,A 0.000,B 0.000,C 90.000,E1 322.924} C_DIS
LIN {X -0.116,Y -597.325,Z 658.587,A 0.000,B 0.000,C 90.000,E1 321.662} C_DIS
LIN {X -0.285,Y -602.312,Z 658.584,A 0.000,B 0.000,C 90.000,E1 321.170} C_DIS
LIN {X -0.208,Y -607.066,Z 658.581,A 0.000,B 0.000,C 90.000,E1 320.642} C_DIS
LIN {X -0.196,Y -612.728,Z 658.578,A 0.000,B 0.000,C 90.000,E1 319.989} C_DIS
LIN {X 0.261,Y -618.038,Z 658.574,A 0.000,B 0.000,C 90.000,E1 319.299} C_DIS
LIN {X -0.105,Y -622.884,Z 658.570,A 0.000,B 0.000,C 90.000,E1 318.690} C_DIS
LIN {X -0.059,Y -628.323,Z 658.566,A 0.000,B 0.000,C 90.000,E1 317.919} C_DIS
LIN {X 0.042,Y -633.501,Z 658.562,A 0.000,B 0.000,C 90.000,E1 317.148} C_DIS
LIN {X -0.210,Y -637.587,Z 658.558,A 0.000,B 0.000,C 90.000,E1 316.539} C_DIS
LIN {X 0.383,Y -643.918,Z 658.553,A 0.000,B 0.000,C 90.000,E1 315.486} C_DIS
LIN {X -0.301,Y -649.155,Z 658.548,A 0.000,B 0.000,C 90.000,E1 314.676} C_DIS
LIN {X 0.008,Y -653.581,Z 658.544,A 0.000,B 0.000,C 90.000,E1 313.905} C_DIS
LIN {X 0.311,Y -659.684,Z 658.538,A 0.000,B 0.000,C 90.000,E1 312.771} C_DIS
LIN {X -0.217,Y -664.704,Z 658.532,A 0.000,B 0.000,C 90.000,E1 311.838} C_DIS
LIN {X -0.188,Y -669.423,Z 658.527,A 0.000,B 0.000,C 90.000,E1 310.862} C_DIS
LIN {X 0.328,Y -672.773,Z 658.523,A 0.000,B 0.000,C 90.000,E1 310.092} C_DIS
LIN {X -0.077,Y -675.798,Z 658.519,A 0.000,B 0.000,C 90.000,E1 309.402} C_DIS
LIN {X 0.065,Y -678.513,Z 658.515,A 0.000,B 0.000,C 90.000,E1 308.669} C_DIS
LIN {X -0.184,Y -681.050,Z 658.511,A 0.000,B 0.000,C 90.000,E1 307.971} C_DIS
LIN {X 0.041,Y -684.130,Z 658.506,A 0.000,B 0.000,C 90.000,E1 306.996} C_DIS
LIN {X 0.436,Y -686.925,Z 658.500,A 0.000,B 0.000,C 90.000,E1 306.011} C_DIS
LIN {X -0.060,Y -690.098,Z 658.494,A 0.000,B 0.000,C 90.000,E1 304.865} C_DIS
LIN {X 0.380,Y -691.903,Z 658.490,A 0.000,B 0.000,C 90.000,E1 304.119} C_DIS
LIN {X -0.115,Y -693.546,Z 658.486,A 0.000,B 0.000,C 90.000,E1 303.452} C_DIS
LIN {X 0.047,Y -696.106,Z 658.479,A 0.000,B 0.000,C 90.000,E1 302.260} C_DIS
LIN {X -0.158,Y -697.935,Z 658.474,A 0.000,B 0.000,C 90.000,E1 301.337} C_DIS
LIN {X 0.025,Y -699.598,Z 658.469,A 0.000,B 0.000,C 90.000,E1 300.384} C_DIS
LIN {X 0.210,Y -700.669,Z 658.465,A 0.000,B 0.000,C 90.000,E1 299.667} C_DIS
LIN {X 0.343,Y -702.230,Z 658.458,A 0.000,B 0.000,C 90.000,E1 298.487} C_DIS
LIN {X -0.111,Y -703.304,Z 658.453,A 0.000,B 0.000,C 90.000,E1 297.590} C_DIS
LIN {X 0.055,Y -704.552,Z 658.447,A 0.000,B 0.000,C 90.000,E1 296.411} C_DIS
LIN {X 0.029,Y -704.783,Z 658.445,A 0.000,B 0.000,C 90.000,E1 296.181} C_DIS
LIN {X -0.028,Y -704.917,Z 658.443,A 0.000,B 0.000,C 90.000,E1 295.720} C_DIS
LIN {X 0.260,Y -704.815,Z 658.442,A 0.000,B 0.000,C 90.000,E1 295.463} C_DIS
LIN {X -0.102,Y -704.170,Z 658.439,A 0.000,B 0.000,C 90.000,E1 295.027} C_DIS
LIN {X 0.184,Y -703.399,Z 658.438,A 0.000,B 0.000,C 90.000,E1 294.771} C_DIS
LIN {X -0.185,Y -700.543,Z 658.435,A 0.000,B 0.000,C 90.000,E1 294.335} C_DIS
LIN {X -0.047,Y -699.694,Z 658.435,A 0.000,B 0.000,C 90.000,E1 294.207} C_DIS
LIN {X 0.089,Y -698.433,Z 658.434,A 0.000,B 0.000,C 90.000,E1 294.079} C_DIS
LIN {X 0.267,Y -696.566,Z 658.433,A 0.000,B 0.000,C 90.000,E1 293.951} C_DIS
LIN {X -0.007,Y -691.405,Z 658.432,A 0.000,B 0.000,C 90.000,E1 293.695} C_DIS
LIN {X -0.378,Y -689.501,Z 658.431,A 0.000,B 0.000,C 90.000,E1 293.643} C_DIS
LIN {X -0.218,Y -682.051,Z 658.430,A 0.000,B 0.000,C 90.000,E1 293.462} C_DIS
LIN {X 0.222,Y -680.099,Z 658.430,A 0.000,B 0.000,C 90.000,E1 293.387} C_DIS
LIN {X 0.216,Y -668.631,Z 658.429,A 0.000,B 0.000,C 90.000,E1 293.259} C_DIS
LIN {X -0.004,Y -658.065,Z 658.429,A 0.000,B 0.000,C 90.000,E1 293.153} C_DIS
LIN {X -0.240,Y -648.519,Z 658.428,A 0.000,B 0.000,C 90.000,E1 293.025} C_DIS
LIN {X 0.212,Y -634.918,Z 658.426,A 0.000,B 0.000,C 90.000,E1 292.717} C_DIS
LIN {X -0.080,Y -625.100,Z 658.425,A 0.000,B 0.000,C 90.000,E1 292.514} C_DIS
LIN {X -0.087,Y -611.676,Z 658.423,A 0.000,B 0.000,C 90.000,E1 292.153} C_DIS
LIN {X 0.073,Y -583.979,Z 658.418,A 0.000,B 0.000,C 90.000,E1 291.280} C_DIS
LIN {X 0.220,Y -576.839,Z 658.417,A 0.000,B 0.000,C 90.000,E1 291.046} C_DIS
LIN {X -0.225,Y -564.346,Z 658.415,A 0.000,B 0.000,C 90.000,E1 290.737} C_DIS
LIN {X -0.174,Y -561.143,Z 658.414,A 0.000,B 0.000,C 90.000,E1 290.610} C_DIS
LIN {X -0.065,Y -556.471,Z 658.413,A 0.000,B 0.000,C 90.000,E1 290.355} C_DIS
LIN {X -0.117,Y -556.401,Z 658.413,A 0.000,B 0.000,C 90.000,E1 290.355} C_DIS
LIN {X 0.001,Y -555.499,Z 658.412,A 0.000,B 0.000,C 90.000,E1 290.174} C_DIS
LIN {X 0.170,Y -554.926,Z 658.410,A 0.000,B 0.000,C 90.000,E1 289.704} C_DIS
LIN {X -0.303,Y -554.681,Z 658.402,A 0.000,B 0.000,C 90.000,E1 288.362} C_DIS
LIN {X 0.226,Y -554.343,Z 658.394,A 0.000,B 0.000,C 90.000,E1 286.913} C_DIS
LIN {X -0.219,Y -554.032,Z 658.388,A 0.000,B 0.000,C 90.000,E1 285.843} C_DIS
LIN {X -0.010,Y -553.428,Z 658.380,A 0.000,B 0.000,C 90.000,E1 284.426} C_DIS
LIN {X 0.192,Y -552.718,Z 658.372,A 0.000,B 0.000,C 90.000,E1 283.008} C_DIS
LIN {X -0.044,Y -551.668,Z 658.362,A 0.000,B 0.000,C 90.000,E1 281.074} C_DIS
LIN {X 0.245,Y -550.829,Z 658.349,A 0.000,B 0.000,C 90.000,E1 278.803} C_DIS
LIN {X -0.202,Y -550.220,Z 658.337,A 0.000,B 0.000,C 90.000,E1 276.606} C_DIS
LIN {X -0.183,Y -549.864,Z 658.324,A 0.000,B 0.000,C 90.000,E1 274.359} C_DIS
LIN {X 0.187,Y -549.564,Z 658.315,A 0.000,B 0.000,C 90.000,E1 272.636} C_DIS
LIN {X -0.083,Y -549.066,Z 658.307,A 0.000,B 0.000,C 90.000,E1 271.260} C_DIS
LIN {X 0.176,Y -548.435,Z 658.299,A 0.000,B 0.000,C 90.000,E1 269.828} C_DIS
LIN {X -0.222,Y -548.049,Z 658.294,A 0.000,B 0.000,C 90.000,E1 269.026} C_DIS
LIN {X 0.117,Y -546.957,Z 658.284,A 0.000,B 0.000,C 90.000,E1 267.020} C_DIS
LIN {X -0.203,Y -546.298,Z 658.277,A 0.000,B 0.000,C 90.000,E1 265.927} C_DIS
LIN {X 0.082,Y -545.017,Z 658.268,A 0.000,B 0.000,C 90.000,E1 264.204} C_DIS
LIN {X 0.265,Y -544.309,Z 658.263,A 0.000,B 0.000,C 90.000,E1 263.337} C_DIS
LIN {X 0.078,Y -542.540,Z 658.254,A 0.000,B 0.000,C 90.000,E1 261.659} C_DIS
LIN {X 0.216,Y -539.498,Z 658.236,A 0.000,B 0.000,C 90.000,E1 258.522} C_DIS
LIN {X 0.166,Y -537.751,Z 658.225,A 0.000,B 0.000,C 90.000,E1 256.533} C_DIS
LIN {X -0.044,Y -537.054,Z 658.221,A 0.000,B 0.000,C 90.000,E1 255.700} C_DIS
LIN {X -0.148,Y -535.830,Z 658.213,A 0.000,B 0.000,C 90.000,E1 254.283} C_DIS
LIN {X 0.059,Y -534.126,Z 658.203,A 0.000,B 0.000,C 90.000,E1 252.543} C_DIS
LIN {X -0.277,Y -532.453,Z 658.194,A 0.000,B 0.000,C 90.000,E1 250.859} C_DIS
LIN {X -0.181,Y -531.138,Z 658.187,A 0.000,B 0.000,C 90.000,E1 249.699} C_DIS
LIN {X 0.081,Y -529.111,Z 658.179,A 0.000,B 0.000,C 90.000,E1 248.230} C_DIS
LIN {X -0.166,Y -527.471,Z 658.173,A 0.000,B 0.000,C 90.000,E1 247.102} C_DIS
LIN {X 0.053,Y -525.639,Z 658.166,A 0.000,B 0.000,C 90.000,E1 245.921} C_DIS
LIN {X 0.142,Y -522.996,Z 658.158,A 0.000,B 0.000,C 90.000,E1 244.460} C_DIS
LIN {X 0.039,Y -520.782,Z 658.152,A 0.000,B 0.000,C 90.000,E1 243.307} C_DIS
LIN {X -0.056,Y -517.206,Z 658.142,A 0.000,B 0.000,C 90.000,E1 241.563} C_DIS
LIN {X 0.101,Y -514.016,Z 658.134,A 0.000,B 0.000,C 90.000,E1 240.078} C_DIS
LIN {X -0.001,Y -510.680,Z 658.126,A 0.000,B 0.000,C 90.000,E1 238.614} C_DIS
LIN {X 0.004,Y -506.737,Z 658.116,A 0.000,B 0.000,C 90.000,E1 236.834} C_DIS
LIN {X 0.116,Y -504.636,Z 658.111,A 0.000,B 0.000,C 90.000,E1 235.928} C_DIS
LIN {X -0.023,Y -500.064,Z 658.101,A 0.000,B 0.000,C 90.000,E1 234.149} C_DIS
LIN {X -0.063,Y -493.943,Z 658.087,A 0.000,B 0.000,C 90.000,E1 231.743} C_DIS
LIN {X 0.046,Y -489.576,Z 658.077,A 0.000,B 0.000,C 90.000,E1 229.908} C_DIS
LIN {X -0.153,Y -486.029,Z 658.069,A 0.000,B 0.000,C 90.000,E1 228.405} C_DIS
LIN {X 0.093,Y -483.103,Z 658.062,A 0.000,B 0.000,C 90.000,E1 227.148} C_DIS
LIN {X -0.257,Y -479.472,Z 658.053,A 0.000,B 0.000,C 90.000,E1 225.648} C_DIS
LIN {X -0.126,Y -474.267,Z 658.041,A 0.000,B 0.000,C 90.000,E1 223.461} C_DIS
LIN {X 0.067,Y -467.889,Z 658.026,A 0.000,B 0.000,C 90.000,E1 220.620} C_DIS
LIN {X -0.110,Y -463.981,Z 658.015,A 0.000,B 0.000,C 90.000,E1 218.749} C_DIS
LIN {X 0.200,Y -461.340,Z 658.008,A 0.000,B 0.000,C 90.000,E1 217.443} C_DIS
LIN {X 0.045,Y -456.906,Z 657.996,A 0.000,B 0.000,C 90.000,E1 215.231} C_DIS
LIN {X 0.062,Y -453.903,Z 657.987,A 0.000,B 0.000,C 90.000,E1 213.627} C_DIS
LIN {X -0.060,Y -449.708,Z 657.974,A 0.000,B 0.000,C 90.000,E1 211.386} C_DIS
LIN {X 0.175,Y -446.154,Z 657.964,A 0.000,B 0.000,C 90.000,E1 209.411} C_DIS
LIN {X 0.168,Y -442.040,Z 657.951,A 0.000,B 0.000,C 90.000,E1 207.129} C_DIS
LIN {X -0.031,Y -439.127,Z 657.942,A 0.000,B 0.000,C 90.000,E1 205.515} C_DIS
LIN {X -0.021,Y -434.973,Z 657.929,A 0.000,B 0.000,C 90.000,E1 203.206} C_DIS
LIN {X 0.117,Y -430.761,Z 657.916,A 0.000,B 0.000,C 90.000,E1 200.865} C_DIS
LIN {X -0.013,Y -426.672,Z 657.903,A 0.000,B 0.000,C 90.000,E1 198.544} C_DIS
LIN {X 0.218,Y -423.300,Z 657.892,A 0.000,B 0.000,C 90.000,E1 196.496} C_DIS
LIN {X 0.130,Y -420.024,Z 657.881,A 0.000,B 0.000,C 90.000,E1 194.481} C_DIS
LIN {X -0.132,Y -416.666,Z 657.869,A 0.000,B 0.000,C 90.000,E1 192.479} C_DIS
LIN {X -0.032,Y -413.004,Z 657.856,A 0.000,B 0.000,C 90.000,E1 190.074} C_DIS
LIN {X 0.118,Y -410.969,Z 657.848,A 0.000,B 0.000,C 90.000,E1 188.681} C_DIS
LIN {X 0.197,Y -408.401,Z 657.839,A 0.000,B 0.000,C 90.000,E1 186.947} C_DIS
LIN {X 0.114,Y -404.144,Z 657.821,A 0.000,B 0.000,C 90.000,E1 183.841} C_DIS
LIN {X -0.144,Y -400.888,Z 657.806,A 0.000,B 0.000,C 90.000,E1 181.088} C_DIS
LIN {X 0.129,Y -397.498,Z 657.785,A 0.000,B 0.000,C 90.000,E1 177.192} C_DIS
LIN {X 0.123,Y -395.810,Z 657.769,A 0.000,B 0.000,C 90.000,E1 174.375} C_DIS
LIN {X 0.153,Y -394.655,Z 657.753,A 0.000,B 0.000,C 90.000,E1 171.546} C_DIS
LIN {X -0.131,Y -394.049,Z 657.737,A 0.000,B 0.000,C 90.000,E1 168.757} C_DIS
LIN {X 0.226,Y -393.822,Z 657.724,A 0.000,B 0.000,C 90.000,E1 166.228} C_DIS
LIN {X -0.085,Y -393.910,Z 657.710,A 0.000,B 0.000,C 90.000,E1 163.795} C_DIS
LIN {X -0.111,Y -394.246,Z 657.694,A 0.000,B 0.000,C 90.000,E1 160.967} C_DIS
LIN {X -0.187,Y -394.539,Z 657.684,A 0.000,B 0.000,C 90.000,E1 159.209} C_DIS
LIN {X -0.079,Y -395.005,Z 657.671,A 0.000,B 0.000,C 90.000,E1 156.719} C_DIS
LIN {X 0.038,Y -395.532,Z 657.657,A 0.000,B 0.000,C 90.000,E1 154.229} C_DIS
LIN {X 0.096,Y -395.993,Z 657.645,A 0.000,B 0.000,C 90.000,E1 152.103} C_DIS
LIN {X 0.007,Y -396.503,Z 657.633,A 0.000,B 0.000,C 90.000,E1 149.999} C_DIS
LIN {X 0.004,Y -397.206,Z 657.620,A 0.000,B 0.000,C 90.000,E1 147.533} C_DIS
LIN {X 0.236,Y -397.968,Z 657.608,A 0.000,B 0.000,C 90.000,E1 145.388} C_DIS
LIN {X -0.160,Y -398.947,Z 657.596,A 0.000,B 0.000,C 90.000,E1 143.336} C_DIS
LIN {X -0.047,Y -399.976,Z 657.585,A 0.000,B 0.000,C 90.000,E1 141.215} C_DIS
LIN {X -0.102,Y -401.340,Z 657.571,A 0.000,B 0.000,C 90.000,E1 138.771} C_DIS
LIN {X -0.231,Y -402.119,Z 657.563,A 0.000,B 0.000,C 90.000,E1 137.391} C_DIS
LIN {X 0.147,Y -403.301,Z 657.552,A 0.000,B 0.000,C 90.000,E1 135.243} C_DIS
LIN {X 0.221,Y -405.302,Z 657.536,A 0.000,B 0.000,C 90.000,E1 132.447} C_DIS
LIN {X 0.018,Y -406.587,Z 657.530,A 0.000,B 0.000,C 90.000,E1 131.434} C_DIS
LIN {X -0.049,Y -408.595,Z 657.526,A 0.000,B 0.000,C 90.000,E1 130.663} C_DIS
LIN {X 0.137,Y -409.868,Z 657.524,A 0.000,B 0.000,C 90.000,E1 130.378} C_DIS
LIN {X -0.247,Y -411.037,Z 657.523,A 0.000,B 0.000,C 90.000,E1 130.172} C_DIS
LIN {X -0.006,Y -413.116,Z 657.522,A 0.000,B 0.000,C 90.000,E1 129.886} C_DIS
LIN {X -0.040,Y -414.335,Z 657.521,A 0.000,B 0.000,C 90.000,E1 129.725} C_DIS
LIN {X -0.042,Y -419.658,Z 657.518,A 0.000,B 0.000,C 90.000,E1 129.241} C_DIS
LIN {X -0.025,Y -424.122,Z 657.516,A 0.000,B 0.000,C 90.000,E1 128.874} C_DIS
LIN {X -0.120,Y -448.111,Z 657.506,A 0.000,B 0.000,C 90.000,E1 127.156} C_DIS
LIN {X 0.101,Y -460.940,Z 657.501,A 0.000,B 0.000,C 90.000,E1 126.217} C_DIS
LIN {X -0.171,Y -471.825,Z 657.497,A 0.000,B 0.000,C 90.000,E1 125.438} C_DIS
LIN {X 0.067,Y -481.021,Z 657.493,A 0.000,B 0.000,C 90.000,E1 124.692} C_DIS
LIN {X 0.135,Y -488.394,Z 657.489,A 0.000,B 0.000,C 90.000,E1 124.072} C_DIS
LIN {X 0.234,Y -497.233,Z 657.485,A 0.000,B 0.000,C 90.000,E1 123.293} C_DIS
LIN {X -0.076,Y -506.992,Z 657.480,A 0.000,B 0.000,C 90.000,E1 122.418} C_DIS
LIN {X 0.164,Y -512.462,Z 657.477,A 0.000,B 0.000,C 90.000,E1 121.878} C_DIS
LIN {X 0.264,Y -521.904,Z 657.472,A 0.000,B 0.000,C 90.000,E1 120.924} C_DIS
LIN {X 0.079,Y -526.871,Z 657.469,A 0.000,B 0.000,C 90.000,E1 120.413} C_DIS
LIN {X -0.144,Y -531.442,Z 657.466,A 0.000,B 0.000,C 90.000,E1 119.922} C_DIS
LIN {X 0.269,Y -536.747,Z 657.462,A 0.000,B 0.000,C 90.000,E1 119.205} C_DIS
LIN {X 0.153,Y -540.737,Z 657.460,A 0.000,B 0.000,C 90.000,E1 118.693} C_DIS
LIN {X 0.230,Y -545.425,Z 657.456,A 0.000,B 0.000,C 90.000,E1 117.975} C_DIS
LIN {X -0.138,Y -549.558,Z 657.452,A 0.000,B 0.000,C 90.000,E1 117.308} C_DIS
LIN {X -0.238,Y -553.237,Z 657.448,A 0.000,B 0.000,C 90.000,E1 116.616} C_DIS
LIN {X -0.055,Y -556.624,Z 657.444,A 0.000,B 0.000,C 90.000,E1 115.899} C_DIS
LIN {X -0.088,Y -559.604,Z 657.440,A 0.000,B 0.000,C 90.000,E1 115.207} C_DIS
LIN {X 0.118,Y -564.018,Z 657.434,A 0.000,B 0.000,C 90.000,E1 114.079} C_DIS
LIN {X -0.135,Y -568.055,Z 657.428,A 0.000,B 0.000,C 90.000,E1 113.003} C_DIS
LIN {X -0.201,Y -569.911,Z 657.425,A 0.000,B 0.000,C 90.000,E1 112.461} C_DIS
LIN {X 0.320,Y -572.452,Z 657.420,A 0.000,B 0.000,C 90.000,E1 111.589} C_DIS
LIN {X 0.125,Y -574.735,Z 657.416,A 0.000,B 0.000,C 90.000,E1 110.791} C_DIS
LIN {X 0.129,Y -577.367,Z 657.410,A 0.000,B 0.000,C 90.000,E1 109.704} C_DIS
LIN {X -0.184,Y -579.841,Z 657.404,A 0.000,B 0.000,C 90.000,E1 108.652} C_DIS
LIN {X 0.100,Y -582.666,Z 657.396,A 0.000,B 0.000,C 90.000,E1 107.275} C_DIS
LIN {X 0.114,Y -586.109,Z 657.387,A 0.000,B 0.000,C 90.000,E1 105.662} C_DIS
LIN {X -0.013,Y -590.635,Z 657.375,A 0.000,B 0.000,C 90.000,E1 103.536} C_DIS
LIN {X 0.180,Y -593.373,Z 657.368,A 0.000,B 0.000,C 90.000,E1 102.187} C_DIS
LIN {X 0.121,Y -596.576,Z 657.359,A 0.000,B 0.000,C 90.000,E1 100.602} C_DIS
LIN {X 0.299,Y -599.226,Z 657.352,A 0.000,B 0.000,C 90.000,E1 99.265} C_DIS
LIN {X 0.216,Y -601.237,Z 657.346,A 0.000,B 0.000,C 90.000,E1 98.219} C_DIS
LIN {X 0.076,Y -603.111,Z 657.340,A 0.000,B 0.000,C 90.000,E1 97.182} C_DIS
LIN {X 0.274,Y -605.298,Z 657.333,A 0.000,B 0.000,C 90.000,E1 95.853} C_DIS
LIN {X 0.101,Y -607.616,Z 657.324,A 0.000,B 0.000,C 90.000,E1 94.302} C_DIS
LIN {X 0.308,Y -609.397,Z 657.317,A 0.000,B 0.000,C 90.000,E1 92.980} C_DIS
LIN {X 0.176,Y -611.058,Z 657.308,A 0.000,B 0.000,C 90.000,E1 91.432} C_DIS
LIN {X -0.222,Y -612.118,Z 657.301,A 0.000,B 0.000,C 90.000,E1 90.172} C_DIS
LIN {X 0.008,Y -612.835,Z 657.294,A 0.000,B 0.000,C 90.000,E1 88.854} C_DIS
LIN {X 0.264,Y -613.254,Z 657.286,A 0.000,B 0.000,C 90.000,E1 87.535} C_DIS
LIN {X 0.237,Y -613.401,Z 657.281,A 0.000,B 0.000,C 90.000,E1 86.502} C_DIS
LIN {X 0.210,Y -613.311,Z 657.275,A 0.000,B 0.000,C 90.000,E1 85.469} C_DIS
LIN {X -0.099,Y -612.982,Z 657.268,A 0.000,B 0.000,C 90.000,E1 84.204} C_DIS
LIN {X -0.078,Y -612.245,Z 657.259,A 0.000,B 0.000,C 90.000,E1 82.648} C_DIS
LIN {X 0.010,Y -611.525,Z 657.253,A 0.000,B 0.000,C 90.000,E1 81.602} C_DIS
LIN {X -0.251,Y -610.757,Z 657.249,A 0.000,B 0.000,C 90.000,E1 80.849} C_DIS
LIN {X -0.177,Y -609.619,Z 657.243,A 0.000,B 0.000,C 90.000,E1 79.803} C_DIS
LIN {X 0.213,Y -608.010,Z 657.236,A 0.000,B 0.000,C 90.000,E1 78.465} C_DIS
LIN {X 0.096,Y -606.151,Z 657.229,A 0.000,B 0.000,C 90.000,E1 77.173} C_DIS
LIN {X -0.051,Y -604.125,Z 657.222,A 0.000,B 0.000,C 90.000,E1 75.880} C_DIS
LIN {X -0.087,Y -601.902,Z 657.214,A 0.000,B 0.000,C 90.000,E1 74.574} C_DIS
LIN {X -0.164,Y -599.499,Z 657.207,A 0.000,B 0.000,C 90.000,E1 73.268} C_DIS
LIN {X -0.112,Y -596.896,Z 657.200,A 0.000,B 0.000,C 90.000,E1 71.945} C_DIS
LIN {X -0.063,Y -595.223,Z 657.195,A 0.000,B 0.000,C 90.000,E1 71.148} C_DIS
LIN {X 0.226,Y -592.821,Z 657.189,A 0.000,B 0.000,C 90.000,E1 70.061} C_DIS
LIN {X -0.084,Y -590.090,Z 657.183,A 0.000,B 0.000,C 90.000,E1 69.028} C_DIS
LIN {X -0.100,Y -587.858,Z 657.179,A 0.000,B 0.000,C 90.000,E1 68.230} C_DIS
LIN {X -0.266,Y -584.549,Z 657.173,A 0.000,B 0.000,C 90.000,E1 67.177} C_DIS
LIN {X -0.113,Y -581.771,Z 657.169,A 0.000,B 0.000,C 90.000,E1 66.357} C_DIS
LIN {X -0.124,Y -577.687,Z 657.163,A 0.000,B 0.000,C 90.000,E1 65.281} C_DIS
LIN {X -0.038,Y -574.467,Z 657.158,A 0.000,B 0.000,C 90.000,E1 64.460} C_DIS
LIN {X 0.011,Y -571.067,Z 657.154,A 0.000,B 0.000,C 90.000,E1 63.640} C_DIS
LIN {X 0.017,Y -567.351,Z 657.149,A 0.000,B 0.000,C 90.000,E1 62.820} C_DIS
LIN {X -0.079,Y -564.759,Z 657.146,A 0.000,B 0.000,C 90.000,E1 62.281} C_DIS
LIN {X -0.056,Y -561.109,Z 657.142,A 0.000,B 0.000,C 90.000,E1 61.591} C_DIS
LIN {X -0.290,Y -557.074,Z 657.138,A 0.000,B 0.000,C 90.000,E1 60.923} C_DIS
LIN {X 0.010,Y -552.521,Z 657.135,A 0.000,B 0.000,C 90.000,E1 60.205} C_DIS
LIN {X -0.035,Y -548.643,Z 657.132,A 0.000,B 0.000,C 90.000,E1 59.665} C_DIS
LIN {X 0.172,Y -543.384,Z 657.128,A 0.000,B 0.000,C 90.000,E1 58.997} C_DIS
LIN {X -0.053,Y -539.806,Z 657.126,A 0.000,B 0.000,C 90.000,E1 58.614} C_DIS
LIN {X 0.060,Y -533.718,Z 657.122,A 0.000,B 0.000,C 90.000,E1 57.995} C_DIS
LIN {X 0.217,Y -529.280,Z 657.120,A 0.000,B 0.000,C 90.000,E1 57.582} C_DIS
LIN {X 0.013,Y -524.637,Z 657.118,A 0.000,B 0.000,C 90.000,E1 57.248} C_DIS
LIN {X -0.125,Y -518.663,Z 657.116,A 0.000,B 0.000,C 90.000,E1 56.834} C_DIS
LIN {X -0.043,Y -512.254,Z 657.113,A 0.000,B 0.000,C 90.000,E1 56.421} C_DIS
LIN {X 0.123,Y -505.456,Z 657.111,A 0.000,B 0.000,C 90.000,E1 56.008} C_DIS
LIN {X 0.129,Y -497.029,Z 657.109,A 0.000,B 0.000,C 90.000,E1 55.548} C_DIS
LIN {X 0.221,Y -477.162,Z 657.103,A 0.000,B 0.000,C 90.000,E1 54.482} C_DIS
LIN {X -0.116,Y -460.373,Z 657.098,A 0.000,B 0.000,C 90.000,E1 53.623} C_DIS
LIN {X 0.025,Y -445.357,Z 657.093,A 0.000,B 0.000,C 90.000,E1 52.763} C_DIS
LIN {X -0.170,Y -433.874,Z 657.089,A 0.000,B 0.000,C 90.000,E1 52.110} C_DIS
LIN {X -0.193,Y -433.863,Z 657.089,A 0.000,B 0.000,C 90.000,E1 52.110} C_DIS
LIN {X -0.167,Y -431.818,Z 657.083,A 0.000,B 0.000,C 90.000,E1 51.009} C_DIS
LIN {X 0.092,Y -431.113,Z 657.081,A 0.000,B 0.000,C 90.000,E1 50.642} C_DIS
LIN {X 0.089,Y -421.963,Z 657.059,A 0.000,B 0.000,C 90.000,E1 46.620} C_DIS
LIN {X 0.024,Y -419.741,Z 657.053,A 0.000,B 0.000,C 90.000,E1 45.445} C_DIS
LIN {X 0.193,Y -419.681,Z 657.051,A 0.000,B 0.000,C 90.000,E1 45.081} C_DIS
LIN {X -0.061,Y -419.834,Z 657.041,A 0.000,B 0.000,C 90.000,E1 43.419} C_DIS
LIN {X -0.229,Y -420.121,Z 657.028,A 0.000,B 0.000,C 90.000,E1 41.067} C_DIS
LIN {X -0.042,Y -420.838,Z 657.015,A 0.000,B 0.000,C 90.000,E1 38.669} C_DIS
LIN {X 0.140,Y -422.270,Z 656.998,A 0.000,B 0.000,C 90.000,E1 35.598} C_DIS
LIN {X 0.110,Y -423.095,Z 656.989,A 0.000,B 0.000,C 90.000,E1 33.913} C_DIS
LIN {X 0.211,Y -423.964,Z 656.979,A 0.000,B 0.000,C 90.000,E1 32.212} C_DIS
LIN {X 0.090,Y -425.015,Z 656.968,A 0.000,B 0.000,C 90.000,E1 30.207} C_DIS
LIN {X -0.222,Y -426.063,Z 656.957,A 0.000,B 0.000,C 90.000,E1 28.231} C_DIS
LIN {X 0.027,Y -427.447,Z 656.944,A 0.000,B 0.000,C 90.000,E1 25.848} C_DIS
LIN {X -0.079,Y -429.946,Z 656.925,A 0.000,B 0.000,C 90.000,E1 22.514} C_DIS
LIN {X -0.069,Y -431.453,Z 656.916,A 0.000,B 0.000,C 90.000,E1 20.844} C_DIS
LIN {X -0.002,Y -432.438,Z 656.908,A 0.000,B 0.000,C 90.000,E1 19.504} C_DIS
LIN {X -0.060,Y -433.275,Z 656.901,A 0.000,B 0.000,C 90.000,E1 18.181} C_DIS
LIN {X -0.178,Y -434.542,Z 656.890,A 0.000,B 0.000,C 90.000,E1 16.205} C_DIS
LIN {X -0.152,Y -436.325,Z 656.877,A 0.000,B 0.000,C 90.000,E1 13.883} C_DIS
LIN {X -0.009,Y -438.064,Z 656.866,A 0.000,B 0.000,C 90.000,E1 11.883} C_DIS
LIN {X -0.129,Y -440.640,Z 656.851,A 0.000,B 0.000,C 90.000,E1 9.265} C_DIS
LIN {X 0.145,Y -443.498,Z 656.837,A 0.000,B 0.000,C 90.000,E1 6.606} C_DIS
LIN {X 0.013,Y -446.669,Z 656.822,A 0.000,B 0.000,C 90.000,E1 4.012} C_DIS
LIN {X 0.004,Y -449.293,Z 656.812,A 0.000,B 0.000,C 90.000,E1 2.064} C_DIS
LIN {X 0.056,Y -453.587,Z 656.795,A 0.000,B 0.000,C 90.000,E1 359.141} C_DIS
LIN {X 0.217,Y -456.794,Z 656.785,A 0.000,B 0.000,C 90.000,E1 357.192} C_DIS
LIN {X -0.217,Y -460.658,Z 656.772,A 0.000,B 0.000,C 90.000,E1 355.008} C_DIS
LIN {X -0.030,Y -463.537,Z 656.763,A 0.000,B 0.000,C 90.000,E1 353.394} C_DIS
LIN {X 0.012,Y -467.003,Z 656.753,A 0.000,B 0.000,C 90.000,E1 351.489} C_DIS
LIN {X 0.190,Y -470.340,Z 656.742,A 0.000,B 0.000,C 90.000,E1 349.577} C_DIS
LIN {X 0.155,Y -473.615,Z 656.732,A 0.000,B 0.000,C 90.000,E1 347.701} C_DIS
LIN {X 0.153,Y -477.598,Z 656.720,A 0.000,B 0.000,C 90.000,E1 345.519} C_DIS
LIN {X 0.087,Y -480.517,Z 656.711,A 0.000,B 0.000,C 90.000,E1 343.976} C_DIS
LIN {X 0.061,Y -484.098,Z 656.701,A 0.000,B 0.000,C 90.000,E1 342.127} C_DIS
LIN {X -0.192,Y -488.304,Z 656.689,A 0.000,B 0.000,C 90.000,E1 340.007} C_DIS
LIN {X -0.091,Y -490.775,Z 656.682,A 0.000,B 0.000,C 90.000,E1 338.773} C_DIS
LIN {X 0.092,Y -493.729,Z 656.674,A 0.000,B 0.000,C 90.000,E1 337.230} C_DIS
LIN {X -0.181,Y -495.907,Z 656.667,A 0.000,B 0.000,C 90.000,E1 336.049} C_DIS
LIN {X -0.166,Y -498.438,Z 656.659,A 0.000,B 0.000,C 90.000,E1 334.537} C_DIS
LIN {X 0.054,Y -500.507,Z 656.652,A 0.000,B 0.000,C 90.000,E1 333.307} C_DIS
LIN {X 0.303,Y -504.386,Z 656.640,A 0.000,B 0.000,C 90.000,E1 331.179} C_DIS
LIN {X -0.075,Y -507.058,Z 656.634,A 0.000,B 0.000,C 90.000,E1 330.177} C_DIS
LIN {X -0.194,Y -508.653,Z 656.632,A 0.000,B 0.000,C 90.000,E1 329.744} C_DIS
LIN {X 0.027,Y -511.798,Z 656.629,A 0.000,B 0.000,C 90.000,E1 329.125} C_DIS
LIN {X -0.072,Y -513.236,Z 656.627,A 0.000,B 0.000,C 90.000,E1 328.918} C_DIS
LIN {X 0.007,Y -515.728,Z 656.626,A 0.000,B 0.000,C 90.000,E1 328.614} C_DIS
LIN {X 0.047,Y -521.580,Z 656.623,A 0.000,B 0.000,C 90.000,E1 328.074} C_DIS
LIN {X 0.109,Y -525.826,Z 656.621,A 0.000,B 0.000,C 90.000,E1 327.709} C_DIS
LIN {X -0.110,Y -537.674,Z 656.616,A 0.000,B 0.000,C 90.000,E1 326.834} C_DIS
LIN {X -0.113,Y -543.405,Z 656.613,A 0.000,B 0.000,C 90.000,E1 326.373} C_DIS
LIN {X -0.267,Y -552.088,Z 656.609,A 0.000,B 0.000,C 90.000,E1 325.674} C_DIS
LIN {X -0.224,Y -556.244,Z 656.607,A 0.000,B 0.000,C 90.000,E1 325.308} C_DIS
LIN {X -0.235,Y -564.550,Z 656.603,A 0.000,B 0.000,C 90.000,E1 324.562} C_DIS
LIN {X -0.045,Y -575.286,Z 656.597,A 0.000,B 0.000,C 90.000,E1 323.543} C_DIS
LIN {X 0.128,Y -584.479,Z 656.593,A 0.000,B 0.000,C 90.000,E1 322.637} C_DIS
LIN {X -0.153,Y -594.618,Z 656.587,A 0.000,B 0.000,C 90.000,E1 321.662} C_DIS
LIN {X 0.035,Y -602.192,Z 656.583,A 0.000,B 0.000,C 90.000,E1 320.884} C_DIS
LIN {X 0.148,Y -606.956,Z 656.580,A 0.000,B 0.000,C 90.000,E1 320.356} C_DIS
LIN {X 0.159,Y -612.670,Z 656.576,A 0.000,B 0.000,C 90.000,E1 319.703} C_DIS
LIN {X -0.200,Y -616.931,Z 656.573,A 0.000,B 0.000,C 90.000,E1 319.218} C_DIS
LIN {X -0.250,Y -621.739,Z 656.570,A 0.000,B 0.000,C 90.000,E1 318.609} C_DIS
LIN {X -0.218,Y -627.245,Z 656.566,A 0.000,B 0.000,C 90.000,E1 317.838} C_DIS
LIN {X -0.172,Y -633.388,Z 656.561,A 0.000,B 0.000,C 90.000,E1 316.944} C_DIS
LIN {X 0.232,Y -641.542,Z 656.554,A 0.000,B 0.000,C 90.000,E1 315.648} C_DIS
LIN {X -0.066,Y -647.730,Z 656.548,A 0.000,B 0.000,C 90.000,E1 314.676} C_DIS
LIN {X 0.195,Y -652.956,Z 656.543,A 0.000,B 0.000,C 90.000,E1 313.785} C_DIS
LIN {X 0.033,Y -658.546,Z 656.538,A 0.000,B 0.000,C 90.000,E1 312.813} C_DIS
LIN {X -0.006,Y -664.287,Z 656.532,A 0.000,B 0.000,C 90.000,E1 311.714} C_DIS
LIN {X -0.037,Y -667.906,Z 656.528,A 0.000,B 0.000,C 90.000,E1 310.987} C_DIS
LIN {X 0.029,Y -672.462,Z 656.522,A 0.000,B 0.000,C 90.000,E1 310.011} C_DIS
LIN {X 0.140,Y -675.467,Z 656.518,A 0.000,B 0.000,C 90.000,E1 309.277} C_DIS
LIN {X 0.285,Y -678.222,Z 656.514,A 0.000,B 0.000,C 90.000,E1 308.543} C_DIS
LIN {X 0.062,Y -681.586,Z 656.509,A 0.000,B 0.000,C 90.000,E1 307.604} C_DIS
LIN {X -0.094,Y -685.318,Z 656.502,A 0.000,B 0.000,C 90.000,E1 306.423} C_DIS
LIN {X -0.084,Y -687.978,Z 656.497,A 0.000,B 0.000,C 90.000,E1 305.471} C_DIS
LIN {X 0.009,Y -691.156,Z 656.490,A 0.000,B 0.000,C 90.000,E1 304.278} C_DIS
LIN {X -0.107,Y -692.856,Z 656.487,A 0.000,B 0.000,C 90.000,E1 303.579} C_DIS
LIN {X -0.331,Y -695.504,Z 656.480,A 0.000,B 0.000,C 90.000,E1 302.418} C_DIS
LIN {X -0.174,Y -697.418,Z 656.475,A 0.000,B 0.000,C 90.000,E1 301.465} C_DIS
LIN {X 0.000,Y -699.160,Z 656.470,A 0.000,B 0.000,C 90.000,E1 300.512} C_DIS
LIN {X -0.163,Y -700.627,Z 656.464,A 0.000,B 0.000,C 90.000,E1 299.589} C_DIS
LIN {X 0.306,Y -701.973,Z 656.459,A 0.000,B 0.000,C 90.000,E1 298.615} C_DIS
LIN {X 0.130,Y -703.392,Z 656.453,A 0.000,B 0.000,C 90.000,E1 297.462} C_DIS
LIN {X -0.016,Y -704.697,Z 656.446,A 0.000,B 0.000,C 90.000,E1 296.309} C_DIS
LIN {X 0.215,Y -704.974,Z 656.442,A 0.000,B 0.000,C 90.000,E1 295.591} C_DIS
LIN {X -0.147,Y -704.358,Z 656.440,A 0.000,B 0.000,C 90.000,E1 295.155} C_DIS
LIN {X 0.140,Y -703.930,Z 656.438,A 0.000,B 0.000,C 90.000,E1 294.899} C_DIS
LIN {X -0.215,Y -702.738,Z 656.437,A 0.000,B 0.000,C 90.000,E1 294.695} C_DIS
LIN {X -0.085,Y -700.593,Z 656.435,A 0.000,B 0.000,C 90.000,E1 294.335} C_DIS
LIN {X 0.053,Y -699.765,Z 656.435,A 0.000,B 0.000,C 90.000,E1 294.207} C_DIS
LIN {X 0.187,Y -698.539,Z 656.434,A 0.000,B 0.000,C 90.000,E1 294.079} C_DIS
LIN {X 0.321,Y -696.650,Z 656.433,A 0.000,B 0.000,C 90.000,E1 293.951} C_DIS
LIN {X 0.296,Y -693.241,Z 656.432,A 0.000,B 0.000,C 90.000,E1 293.770} C_DIS
LIN {X -0.155,Y -689.495,Z 656.431,A 0.000,B 0.000,C 90.000,E1 293.643} C_DIS
LIN {X -0.073,Y -686.857,Z 656.431,A 0.000,B 0.000,C 90.000,E1 293.567} C_DIS
LIN {X 0.353,Y -679.886,Z 656.430,A 0.000,B 0.000,C 90.000,E1 293.387} C_DIS
LIN {X 0.298,Y -667.867,Z 656.429,A 0.000,B 0.000,C 90.000,E1 293.259} C_DIS
LIN {X -0.235,Y -659.238,Z 656.429,A 0.000,B 0.000,C 90.000,E1 293.206} C_DIS
LIN {X 0.133,Y -649.447,Z 656.428,A 0.000,B 0.000,C 90.000,E1 293.025} C_DIS
LIN {X 0.115,Y -639.747,Z 656.427,A 0.000,B 0.000,C 90.000,E1 292.845} C_DIS
LIN {X -0.087,Y -629.481,Z 656.426,A 0.000,B 0.000,C 90.000,E1 292.642} C_DIS
LIN {X 0.116,Y -616.211,Z 656.424,A 0.000,B 0.000,C 90.000,E1 292.280} C_DIS
LIN {X 0.176,Y -595.944,Z 656.420,A 0.000,B 0.000,C 90.000,E1 291.663} C_DIS
LIN {X 0.289,Y -578.402,Z 656.417,A 0.000,B 0.000,C 90.000,E1 291.099} C_DIS
LIN {X -0.187,Y -563.990,Z 656.415,A 0.000,B 0.000,C 90.000,E1 290.737} C_DIS
LIN {X 0.084,Y -561.476,Z 656.415,A 0.000,B 0.000,C 90.000,E1 290.610} C_DIS
LIN {X -0.285,Y -557.215,Z 656.413,A 0.000,B 0.000,C 90.000,E1 290.429} C_DIS
LIN {X -0.038,Y -556.440,Z 656.413,A 0.000,B 0.000,C 90.000,E1 290.355} C_DIS
LIN {X -0.080,Y -556.387,Z 656.413,A 0.000,B 0.000,C 90.000,E1 290.355} C_DIS
LIN {X 0.056,Y -555.574,Z 656.412,A 0.000,B 0.000,C 90.000,E1 290.194} C_DIS
LIN {X -0.147,Y -555.024,Z 656.410,A 0.000,B 0.000,C 90.000,E1 289.758} C_DIS
LIN {X -0.133,Y -554.777,Z 656.402,A 0.000,B 0.000,C 90.000,E1 288.362} C_DIS
LIN {X 0.121,Y -554.539,Z 656.396,A 0.000,B 0.000,C 90.000,E1 287.221} C_DIS
LIN {X -0.046,Y -554.132,Z 656.388,A 0.000,B 0.000,C 90.000,E1 285.843} C_DIS
LIN {X 0.165,Y -553.530,Z 656.380,A 0.000,B 0.000,C 90.000,E1 284.426} C_DIS
LIN {X -0.170,Y -552.820,Z 656.372,A 0.000,B 0.000,C 90.000,E1 283.063} C_DIS
LIN {X 0.134,Y -551.772,Z 656.362,A 0.000,B 0.000,C 90.000,E1 281.074} C_DIS
LIN {X -0.118,Y -550.928,Z 656.349,A 0.000,B 0.000,C 90.000,E1 278.859} C_DIS
LIN {X -0.018,Y -550.318,Z 656.337,A 0.000,B 0.000,C 90.000,E1 276.606} C_DIS
LIN {X 0.004,Y -549.931,Z 656.324,A 0.000,B 0.000,C 90.000,E1 274.359} C_DIS
LIN {X -0.175,Y -549.619,Z 656.315,A 0.000,B 0.000,C 90.000,E1 272.694} C_DIS
LIN {X 0.158,Y -549.028,Z 656.306,A 0.000,B 0.000,C 90.000,E1 270.974} C_DIS
LIN {X -0.082,Y -548.244,Z 656.296,A 0.000,B 0.000,C 90.000,E1 269.312} C_DIS
LIN {X 0.265,Y -547.190,Z 656.285,A 0.000,B 0.000,C 90.000,E1 267.306} C_DIS
LIN {X -0.012,Y -546.376,Z 656.277,A 0.000,B 0.000,C 90.000,E1 265.927} C_DIS
LIN {X 0.168,Y -545.532,Z 656.271,A 0.000,B 0.000,C 90.000,E1 264.780} C_DIS
LIN {X -0.164,Y -544.659,Z 656.265,A 0.000,B 0.000,C 90.000,E1 263.685} C_DIS
LIN {X 0.030,Y -543.564,Z 656.259,A 0.000,B 0.000,C 90.000,E1 262.534} C_DIS
LIN {X -0.182,Y -542.039,Z 656.251,A 0.000,B 0.000,C 90.000,E1 261.141} C_DIS
LIN {X -0.114,Y -539.609,Z 656.237,A 0.000,B 0.000,C 90.000,E1 258.578} C_DIS
LIN {X -0.156,Y -537.857,Z 656.225,A 0.000,B 0.000,C 90.000,E1 256.589} C_DIS
LIN {X 0.159,Y -537.162,Z 656.221,A 0.000,B 0.000,C 90.000,E1 255.700} C_DIS
LIN {X 0.055,Y -535.938,Z 656.213,A 0.000,B 0.000,C 90.000,E1 254.283} C_DIS
LIN {X 0.264,Y -534.232,Z 656.203,A 0.000,B 0.000,C 90.000,E1 252.543} C_DIS
LIN {X -0.070,Y -532.592,Z 656.194,A 0.000,B 0.000,C 90.000,E1 250.859} C_DIS
LIN {X 0.028,Y -531.276,Z 656.187,A 0.000,B 0.000,C 90.000,E1 249.699} C_DIS
LIN {X 0.105,Y -529.657,Z 656.181,A 0.000,B 0.000,C 90.000,E1 248.539} C_DIS
LIN {X 0.046,Y -527.589,Z 656.173,A 0.000,B 0.000,C 90.000,E1 247.102} C_DIS
LIN {X 0.265,Y -525.746,Z 656.166,A 0.000,B 0.000,C 90.000,E1 245.921} C_DIS
LIN {X 0.129,Y -523.078,Z 656.158,A 0.000,B 0.000,C 90.000,E1 244.485} C_DIS
LIN {X 0.019,Y -520.855,Z 656.152,A 0.000,B 0.000,C 90.000,E1 243.332} C_DIS
LIN {X 0.157,Y -517.263,Z 656.142,A 0.000,B 0.000,C 90.000,E1 241.563} C_DIS
LIN {X -0.042,Y -514.744,Z 656.136,A 0.000,B 0.000,C 90.000,E1 240.411} C_DIS
LIN {X 0.226,Y -512.073,Z 656.129,A 0.000,B 0.000,C 90.000,E1 239.203} C_DIS
LIN {X -0.108,Y -507.431,Z 656.118,A 0.000,B 0.000,C 90.000,E1 237.168} C_DIS
LIN {X 0.045,Y -504.665,Z 656.111,A 0.000,B 0.000,C 90.000,E1 235.960} C_DIS
LIN {X -0.216,Y -500.057,Z 656.101,A 0.000,B 0.000,C 90.000,E1 234.196} C_DIS
LIN {X 0.146,Y -493.930,Z 656.088,A 0.000,B 0.000,C 90.000,E1 231.743} C_DIS
LIN {X -0.128,Y -490.995,Z 656.081,A 0.000,B 0.000,C 90.000,E1 230.561} C_DIS
LIN {X 0.226,Y -486.706,Z 656.071,A 0.000,B 0.000,C 90.000,E1 228.690} C_DIS
LIN {X -0.032,Y -483.085,Z 656.062,A 0.000,B 0.000,C 90.000,E1 227.187} C_DIS
LIN {X -0.056,Y -479.443,Z 656.054,A 0.000,B 0.000,C 90.000,E1 225.648} C_DIS
LIN {X 0.072,Y -474.248,Z 656.042,A 0.000,B 0.000,C 90.000,E1 223.461} C_DIS
LIN {X -0.164,Y -468.572,Z 656.028,A 0.000,B 0.000,C 90.000,E1 220.987} C_DIS
LIN {X 0.083,Y -463.924,Z 656.015,A 0.000,B 0.000,C 90.000,E1 218.749} C_DIS
LIN {X -0.255,Y -461.266,Z 656.008,A 0.000,B 0.000,C 90.000,E1 217.523} C_DIS
LIN {X 0.232,Y -456.862,Z 655.996,A 0.000,B 0.000,C 90.000,E1 215.231} C_DIS
LIN {X -0.003,Y -453.857,Z 655.987,A 0.000,B 0.000,C 90.000,E1 213.658} C_DIS
LIN {X 0.122,Y -449.692,Z 655.974,A 0.000,B 0.000,C 90.000,E1 211.386} C_DIS
LIN {X 0.034,Y -445.590,Z 655.962,A 0.000,B 0.000,C 90.000,E1 209.127} C_DIS
LIN {X -0.046,Y -442.033,Z 655.951,A 0.000,B 0.000,C 90.000,E1 207.180} C_DIS
LIN {X 0.117,Y -439.697,Z 655.944,A 0.000,B 0.000,C 90.000,E1 205.848} C_DIS
LIN {X 0.080,Y -436.685,Z 655.935,A 0.000,B 0.000,C 90.000,E1 204.207} C_DIS
LIN {X -0.016,Y -434.327,Z 655.927,A 0.000,B 0.000,C 90.000,E1 202.898} C_DIS
LIN {X 0.106,Y -430.146,Z 655.914,A 0.000,B 0.000,C 90.000,E1 200.556} C_DIS
LIN {X 0.158,Y -426.674,Z 655.903,A 0.000,B 0.000,C 90.000,E1 198.544} C_DIS
LIN {X -0.017,Y -423.296,Z 655.892,A 0.000,B 0.000,C 90.000,E1 196.551} C_DIS
LIN {X -0.109,Y -420.027,Z 655.881,A 0.000,B 0.000,C 90.000,E1 194.537} C_DIS
LIN {X -0.020,Y -417.273,Z 655.871,A 0.000,B 0.000,C 90.000,E1 192.827} C_DIS
LIN {X 0.135,Y -413.042,Z 655.856,A 0.000,B 0.000,C 90.000,E1 190.074} C_DIS
LIN {X -0.184,Y -411.018,Z 655.849,A 0.000,B 0.000,C 90.000,E1 188.746} C_DIS
LIN {X -0.070,Y -407.928,Z 655.837,A 0.000,B 0.000,C 90.000,E1 186.663} C_DIS
LIN {X -0.117,Y -404.627,Z 655.824,A 0.000,B 0.000,C 90.000,E1 184.245} C_DIS
LIN {X 0.104,Y -401.710,Z 655.810,A 0.000,B 0.000,C 90.000,E1 181.776} C_DIS
LIN {X 0.051,Y -398.370,Z 655.791,A 0.000,B 0.000,C 90.000,E1 178.282} C_DIS
LIN {X -0.065,Y -396.084,Z 655.771,A 0.000,B 0.000,C 90.000,E1 174.780} C_DIS
LIN {X -0.030,Y -394.875,Z 655.755,A 0.000,B 0.000,C 90.000,E1 171.951} C_DIS
LIN {X 0.085,Y -394.238,Z 655.740,A 0.000,B 0.000,C 90.000,E1 169.106} C_DIS
LIN {X 0.025,Y -393.974,Z 655.724,A 0.000,B 0.000,C 90.000,E1 166.284} C_DIS
LIN {X 0.101,Y -394.090,Z 655.710,A 0.000,B 0.000,C 90.000,E1 163.795} C_DIS
LIN {X 0.081,Y -394.420,Z 655.694,A 0.000,B 0.000,C 90.000,E1 160.967} C_DIS
LIN {X 0.008,Y -394.709,Z 655.685,A 0.000,B 0.000,C 90.000,E1 159.209} C_DIS
LIN {X -0.035,Y -395.210,Z 655.671,A 0.000,B 0.000,C 90.000,E1 156.741} C_DIS
LIN {X -0.112,Y -395.757,Z 655.657,A 0.000,B 0.000,C 90.000,E1 154.280} C_DIS
LIN {X -0.042,Y -396.211,Z 655.645,A 0.000,B 0.000,C 90.000,E1 152.153} C_DIS
LIN {X 0.226,Y -396.753,Z 655.634,A 0.000,B 0.000,C 90.000,E1 149.999} C_DIS
LIN {X -0.230,Y -397.581,Z 655.618,A 0.000,B 0.000,C 90.000,E1 147.248} C_DIS
LIN {X -0.137,Y -398.847,Z 655.600,A 0.000,B 0.000,C 90.000,E1 144.069} C_DIS
LIN {X -0.034,Y -399.823,Z 655.589,A 0.000,B 0.000,C 90.000,E1 141.949} C_DIS
LIN {X 0.100,Y -400.874,Z 655.577,A 0.000,B 0.000,C 90.000,E1 139.828} C_DIS
LIN {X 0.083,Y -401.835,Z 655.567,A 0.000,B 0.000,C 90.000,E1 138.081} C_DIS
LIN {X 0.178,Y -402.990,Z 655.556,A 0.000,B 0.000,C 90.000,E1 135.972} C_DIS
LIN {X 0.075,Y -404.931,Z 655.538,A 0.000,B 0.000,C 90.000,E1 132.852} C_DIS
LIN {X 0.007,Y -406.333,Z 655.530,A 0.000,B 0.000,C 90.000,E1 131.472} C_DIS
LIN {X -0.160,Y -406.998,Z 655.529,A 0.000,B 0.000,C 90.000,E1 131.148} C_DIS
LIN {X -0.095,Y -408.644,Z 655.525,A 0.000,B 0.000,C 90.000,E1 130.458} C_DIS
LIN {X 0.039,Y -410.064,Z 655.523,A 0.000,B 0.000,C 90.000,E1 130.092} C_DIS
LIN {X -0.042,Y -411.142,Z 655.522,A 0.000,B 0.000,C 90.000,E1 129.930} C_DIS
LIN {X 0.119,Y -413.581,Z 655.520,A 0.000,B 0.000,C 90.000,E1 129.564} C_DIS
LIN {X -0.037,Y -418.514,Z 655.517,A 0.000,B 0.000,C 90.000,E1 129.116} C_DIS
LIN {X 0.149,Y -422.654,Z 655.515,A 0.000,B 0.000,C 90.000,E1 128.749} C_DIS
LIN {X 0.043,Y -435.690,Z 655.510,A 0.000,B 0.000,C 90.000,E1 127.810} C_DIS
LIN {X 0.190,Y -450.117,Z 655.505,A 0.000,B 0.000,C 90.000,E1 126.790} C_DIS
LIN {X 0.062,Y -461.355,Z 655.500,A 0.000,B 0.000,C 90.000,E1 126.011} C_DIS
LIN {X 0.062,Y -469.138,Z 655.497,A 0.000,B 0.000,C 90.000,E1 125.438} C_DIS
LIN {X -0.046,Y -478.409,Z 655.493,A 0.000,B 0.000,C 90.000,E1 124.739} C_DIS
LIN {X -0.245,Y -482.969,Z 655.491,A 0.000,B 0.000,C 90.000,E1 124.405} C_DIS
LIN {X -0.236,Y -488.866,Z 655.488,A 0.000,B 0.000,C 90.000,E1 123.913} C_DIS
LIN {X 0.062,Y -497.706,Z 655.484,A 0.000,B 0.000,C 90.000,E1 123.118} C_DIS
LIN {X 0.049,Y -508.874,Z 655.478,A 0.000,B 0.000,C 90.000,E1 122.084} C_DIS
LIN {X 0.146,Y -514.466,Z 655.475,A 0.000,B 0.000,C 90.000,E1 121.544} C_DIS
LIN {X 0.102,Y -521.312,Z 655.472,A 0.000,B 0.000,C 90.000,E1 120.875} C_DIS
LIN {X -0.079,Y -527.762,Z 655.468,A 0.000,B 0.000,C 90.000,E1 120.207} C_DIS
LIN {X -0.166,Y -531.568,Z 655.465,A 0.000,B 0.000,C 90.000,E1 119.795} C_DIS
LIN {X -0.176,Y -537.333,Z 655.461,A 0.000,B 0.000,C 90.000,E1 119.077} C_DIS
LIN {X 0.138,Y -540.618,Z 655.459,A 0.000,B 0.000,C 90.000,E1 118.615} C_DIS
LIN {X 0.085,Y -544.534,Z 655.456,A 0.000,B 0.000,C 90.000,E1 118.052} C_DIS
LIN {X -0.106,Y -549.428,Z 655.451,A 0.000,B 0.000,C 90.000,E1 117.257} C_DIS
LIN {X 0.043,Y -553.162,Z 655.448,A 0.000,B 0.000,C 90.000,E1 116.539} C_DIS
LIN {X -0.021,Y -556.620,Z 655.444,A 0.000,B 0.000,C 90.000,E1 115.848} C_DIS
LIN {X -0.153,Y -560.213,Z 655.439,A 0.000,B 0.000,C 90.000,E1 115.027} C_DIS
LIN {X 0.063,Y -564.665,Z 655.433,A 0.000,B 0.000,C 90.000,E1 113.898} C_DIS
LIN {X 0.008,Y -567.750,Z 655.428,A 0.000,B 0.000,C 90.000,E1 113.078} C_DIS
LIN {X -0.238,Y -570.532,Z 655.424,A 0.000,B 0.000,C 90.000,E1 112.280} C_DIS
LIN {X 0.292,Y -573.052,Z 655.419,A 0.000,B 0.000,C 90.000,E1 111.408} C_DIS
LIN {X -0.263,Y -574.656,Z 655.416,A 0.000,B 0.000,C 90.000,E1 110.918} C_DIS
LIN {X -0.064,Y -577.378,Z 655.410,A 0.000,B 0.000,C 90.000,E1 109.812} C_DIS
LIN {X -0.021,Y -579.926,Z 655.404,A 0.000,B 0.000,C 90.000,E1 108.725} C_DIS
LIN {X -0.282,Y -582.795,Z 655.397,A 0.000,B 0.000,C 90.000,E1 107.402} C_DIS
LIN {X -0.261,Y -586.231,Z 655.388,A 0.000,B 0.000,C 90.000,E1 105.788} C_DIS
LIN {X -0.238,Y -590.822,Z 655.376,A 0.000,B 0.000,C 90.000,E1 103.647} C_DIS
LIN {X -0.049,Y -593.619,Z 655.368,A 0.000,B 0.000,C 90.000,E1 102.299} C_DIS
LIN {X 0.189,Y -596.334,Z 655.361,A 0.000,B 0.000,C 90.000,E1 100.950} C_DIS
LIN {X 0.067,Y -599.586,Z 655.352,A 0.000,B 0.000,C 90.000,E1 99.378} C_DIS
LIN {X 0.203,Y -602.126,Z 655.345,A 0.000,B 0.000,C 90.000,E1 98.049} C_DIS
LIN {X 0.153,Y -603.968,Z 655.339,A 0.000,B 0.000,C 90.000,E1 97.004} C_DIS
LIN {X 0.048,Y -605.784,Z 655.333,A 0.000,B 0.000,C 90.000,E1 95.967} C_DIS
LIN {X 0.146,Y -608.484,Z 655.323,A 0.000,B 0.000,C 90.000,E1 94.131} C_DIS
LIN {X 0.094,Y -609.950,Z 655.317,A 0.000,B 0.000,C 90.000,E1 93.094} C_DIS
LIN {X -0.028,Y -611.619,Z 655.309,A 0.000,B 0.000,C 90.000,E1 91.547} C_DIS
LIN {X 0.224,Y -612.327,Z 655.304,A 0.000,B 0.000,C 90.000,E1 90.745} C_DIS
LIN {X 0.167,Y -613.047,Z 655.299,A 0.000,B 0.000,C 90.000,E1 89.714} C_DIS
LIN {X -0.176,Y -613.524,Z 655.294,A 0.000,B 0.000,C 90.000,E1 88.969} C_DIS
LIN {X -0.227,Y -613.993,Z 655.286,A 0.000,B 0.000,C 90.000,E1 87.421} C_DIS
LIN {X -0.245,Y -614.077,Z 655.280,A 0.000,B 0.000,C 90.000,E1 86.388} C_DIS
LIN {X -0.265,Y -613.924,Z 655.274,A 0.000,B 0.000,C 90.000,E1 85.355} C_DIS
LIN {X -0.238,Y -613.689,Z 655.268,A 0.000,B 0.000,C 90.000,E1 84.318} C_DIS
LIN {X -0.198,Y -612.908,Z 655.260,A 0.000,B 0.000,C 90.000,E1 82.761} C_DIS
LIN {X -0.186,Y -612.186,Z 655.254,A 0.000,B 0.000,C 90.000,E1 81.724} C_DIS
LIN {X -0.094,Y -611.717,Z 655.251,A 0.000,B 0.000,C 90.000,E1 81.197} C_DIS
LIN {X 0.338,Y -610.288,Z 655.244,A 0.000,B 0.000,C 90.000,E1 79.859} C_DIS
LIN {X 0.144,Y -608.652,Z 655.237,A 0.000,B 0.000,C 90.000,E1 78.578} C_DIS
LIN {X 0.045,Y -606.751,Z 655.229,A 0.000,B 0.000,C 90.000,E1 77.285} C_DIS
LIN {X -0.086,Y -604.734,Z 655.222,A 0.000,B 0.000,C 90.000,E1 75.992} C_DIS
LIN {X -0.105,Y -602.475,Z 655.215,A 0.000,B 0.000,C 90.000,E1 74.685} C_DIS
LIN {X -0.164,Y -600.067,Z 655.208,A 0.000,B 0.000,C 90.000,E1 73.378} C_DIS
LIN {X -0.095,Y -597.446,Z 655.200,A 0.000,B 0.000,C 90.000,E1 72.054} C_DIS
LIN {X 0.228,Y -595.107,Z 655.194,A 0.000,B 0.000,C 90.000,E1 70.967} C_DIS
LIN {X -0.044,Y -592.623,Z 655.189,A 0.000,B 0.000,C 90.000,E1 69.934} C_DIS
LIN {X 0.197,Y -589.764,Z 655.183,A 0.000,B 0.000,C 90.000,E1 68.847} C_DIS
LIN {X 0.175,Y -587.425,Z 655.178,A 0.000,B 0.000,C 90.000,E1 68.050} C_DIS
LIN {X -0.187,Y -584.882,Z 655.174,A 0.000,B 0.000,C 90.000,E1 67.283} C_DIS
LIN {X -0.257,Y -582.054,Z 655.169,A 0.000,B 0.000,C 90.000,E1 66.485} C_DIS
LIN {X 0.260,Y -577.954,Z 655.163,A 0.000,B 0.000,C 90.000,E1 65.357} C_DIS
LIN {X -0.176,Y -574.745,Z 655.159,A 0.000,B 0.000,C 90.000,E1 64.588} C_DIS
LIN {X -0.123,Y -571.266,Z 655.154,A 0.000,B 0.000,C 90.000,E1 63.768} C_DIS
LIN {X -0.113,Y -567.483,Z 655.150,A 0.000,B 0.000,C 90.000,E1 62.948} C_DIS
LIN {X 0.198,Y -564.124,Z 655.146,A 0.000,B 0.000,C 90.000,E1 62.231} C_DIS
LIN {X 0.065,Y -560.400,Z 655.142,A 0.000,B 0.000,C 90.000,E1 61.563} C_DIS
LIN {X 0.042,Y -556.203,Z 655.138,A 0.000,B 0.000,C 90.000,E1 60.873} C_DIS
LIN {X 0.110,Y -552.644,Z 655.135,A 0.000,B 0.000,C 90.000,E1 60.333} C_DIS
LIN {X -0.073,Y -548.598,Z 655.132,A 0.000,B 0.000,C 90.000,E1 59.793} C_DIS
LIN {X 0.188,Y -543.997,Z 655.129,A 0.000,B 0.000,C 90.000,E1 59.203} C_DIS
LIN {X -0.034,Y -538.948,Z 655.126,A 0.000,B 0.000,C 90.000,E1 58.663} C_DIS
LIN {X 0.031,Y -533.394,Z 655.123,A 0.000,B 0.000,C 90.000,E1 58.122} C_DIS
LIN {X 0.037,Y -529.012,Z 655.121,A 0.000,B 0.000,C 90.000,E1 57.740} C_DIS
LIN {X 0.056,Y -524.236,Z 655.119,A 0.000,B 0.000,C 90.000,E1 57.375} C_DIS
LIN {X 0.200,Y -517.839,Z 655.116,A 0.000,B 0.000,C 90.000,E1 56.914} C_DIS
LIN {X 0.244,Y -511.182,Z 655.114,A 0.000,B 0.000,C 90.000,E1 56.501} C_DIS
LIN {X 0.093,Y -504.491,Z 655.112,A 0.000,B 0.000,C 90.000,E1 56.135} C_DIS
LIN {X 0.135,Y -495.941,Z 655.109,A 0.000,B 0.000,C 90.000,E1 55.674} C_DIS
LIN {X 0.287,Y -477.720,Z 655.104,A 0.000,B 0.000,C 90.000,E1 54.689} C_DIS
LIN {X -0.032,Y -460.847,Z 655.099,A 0.000,B 0.000,C 90.000,E1 53.829} C_DIS
LIN {X -0.110,Y -445.908,Z 655.094,A 0.000,B 0.000,C 90.000,E1 53.004} C_DIS
